C03679=1100.327,-122.776,-46.976,-179.986,4.175,148.668
C03680=1100.332,-123.026,-46.967,-179.985,4.170,148.666
C03681=1100.338,-123.276,-46.957,-179.985,4.164,148.665
C03682=1100.343,-123.525,-46.946,-179.984,4.159,148.663
C03683=1100.348,-123.775,-46.938,-179.983,4.153,148.662
C03684=1100.353,-124.026,-46.927,-179.983,4.148,148.661
C03685=1100.358,-124.275,-46.917,-179.982,4.143,148.659
C03686=1100.364,-124.524,-46.907,-179.982,4.138,148.658
C03687=1100.369,-124.774,-46.898,-179.981,4.133,148.657
C03688=1100.375,-125.024,-46.888,-179.980,4.128,148.655
C03689=1100.380,-125.274,-46.877,-179.980,4.122,148.654
C03690=1100.385,-125.524,-46.869,-179.979,4.117,148.653
C03691=1100.390,-125.773,-46.858,-179.978,4.111,148.651
C03692=1100.395,-126.023,-46.849,-179.978,4.106,148.650
C03693=1100.401,-126.273,-46.839,-179.977,4.102,148.649
C03694=1100.406,-126.522,-46.830,-179.976,4.096,148.647
C03695=1100.410,-126.736,-46.821,-179.976,4.091,148.646
C03696=1100.415,-126.951,-46.813,-179.975,4.087,148.645
C03697=1100.419,-127.165,-46.805,-179.974,4.083,148.644
C03698=1100.424,-127.380,-46.796,-179.974,4.077,148.642
C03699=1100.428,-127.594,-46.788,-179.973,4.073,148.641
C03700=1100.433,-127.809,-46.780,-179.972,4.069,148.640
C03701=1100.437,-128.023,-46.771,-179.972,4.064,148.639
C03702=1100.442,-128.238,-46.763,-179.971,4.059,148.637
C03703=1100.019,-128.228,-46.789,-179.964,4.064,148.636
C03704=1100.015,-128.014,-46.798,-179.965,4.068,148.637
C03705=1100.010,-127.799,-46.806,-179.966,4.073,148.639
C03706=1100.006,-127.585,-46.814,-179.966,4.078,148.640
C03707=1100.001,-127.371,-46.823,-179.966,4.082,148.641
C03708=1099.997,-127.156,-46.831,-179.967,4.086,148.642
C03709=1099.992,-126.942,-46.839,-179.968,4.091,148.643
C03710=1099.987,-126.728,-46.847,-179.968,4.096,148.645
C03711=1099.983,-126.513,-46.856,-179.969,4.100,148.646
C03712=1099.978,-126.263,-46.866,-179.970,4.105,148.647
C03713=1099.972,-126.013,-46.875,-179.970,4.111,148.649
C03714=1099.967,-125.764,-46.885,-179.971,4.116,148.650
C03715=1099.962,-125.515,-46.895,-179.972,4.121,148.651
C03716=1099.956,-125.264,-46.904,-179.972,4.127,148.653
C03717=1099.952,-125.014,-46.914,-179.973,4.131,148.654
C03718=1099.946,-124.765,-46.925,-179.974,4.137,148.655
C03719=1099.941,-124.515,-46.933,-179.974,4.142,148.657
C03720=1099.935,-124.266,-46.944,-179.975,4.147,148.658
C03721=1099.930,-124.016,-46.954,-179.976,4.153,148.660
C03722=1099.926,-123.766,-46.964,-179.976,4.158,148.661
C03723=1099.920,-123.516,-46.973,-179.977,4.164,148.662
C03724=1099.915,-123.267,-46.983,-179.978,4.168,148.663
C03725=1099.909,-123.017,-46.993,-179.979,4.173,148.665
C03726=1099.904,-122.766,-47.003,-179.979,4.179,148.666
C03727=1099.899,-122.517,-47.013,-179.980,4.184,148.668
C03728=1099.894,-122.267,-47.023,-179.980,4.189,148.669
C03729=1099.888,-122.018,-47.033,-179.982,4.194,148.670
C03730=1099.884,-121.768,-47.043,-179.982,4.199,148.672
C03731=1099.878,-121.518,-47.053,-179.983,4.205,148.673
C03732=1099.873,-121.269,-47.062,-179.983,4.210,148.674
C03733=1099.867,-121.019,-47.072,-179.984,4.215,148.676
C03734=1099.862,-120.769,-47.083,-179.984,4.220,148.677
C03735=1099.857,-120.520,-47.093,-179.985,4.225,148.678
C03736=1099.852,-120.269,-47.102,-179.986,4.230,148.680
C03737=1099.846,-120.020,-47.112,-179.986,4.235,148.681
C03738=1099.842,-119.770,-47.122,-179.987,4.241,148.682
C03739=1099.836,-119.520,-47.132,-179.987,4.246,148.683
C03740=1099.830,-119.271,-47.143,-179.988,4.251,148.685
C03741=1099.826,-119.021,-47.153,-179.989,4.256,148.686
C03742=1099.820,-118.771,-47.162,-179.989,4.261,148.687
C03743=1099.815,-118.521,-47.172,-179.990,4.267,148.689
C03744=1099.810,-118.271,-47.183,-179.991,4.271,148.690
C03745=1099.805,-118.022,-47.193,-179.991,4.277,148.692
C03746=1099.799,-117.772,-47.203,-179.992,4.282,148.693
C03747=1099.794,-117.523,-47.213,-179.992,4.287,148.694
C03748=1099.789,-117.272,-47.224,-179.993,4.292,148.695
C03749=1099.784,-117.023,-47.233,-179.994,4.297,148.697
C03750=1099.778,-116.774,-47.243,-179.994,4.302,148.698
C03751=1099.773,-116.523,-47.253,-179.995,4.307,148.699
C03752=1099.767,-116.273,-47.263,-179.995,4.313,148.701
C03753=1099.762,-116.024,-47.273,-179.996,4.317,148.702
C03754=1099.757,-115.774,-47.284,-179.997,4.322,148.703
C03755=1099.752,-115.524,-47.294,-179.997,4.328,148.704
C03756=1099.746,-115.275,-47.304,-179.997,4.333,148.706
C03757=1099.742,-115.025,-47.314,-179.998,4.337,148.707
C03758=1099.736,-114.775,-47.324,-179.999,4.343,148.708
C03759=1099.731,-114.526,-47.334,-179.999,4.348,148.710
C03760=1099.727,-114.312,-47.343,-180.000,4.352,148.711
C03761=1099.722,-114.097,-47.352,180.000,4.356,148.712
C03762=1099.717,-113.882,-47.361,180.000,4.361,148.713
C03763=1099.713,-113.668,-47.370,179.999,4.365,148.714
C03764=1099.709,-113.454,-47.378,179.998,4.369,148.715
C03765=1099.705,-113.240,-47.387,179.998,4.374,148.716
C03766=1099.700,-113.025,-47.396,179.997,4.378,148.717
C03767=1099.695,-112.811,-47.405,179.997,4.383,148.718
C03768=1099.690,-112.562,-47.415,179.996,4.387,148.720
C03769=1099.685,-112.312,-47.426,179.996,4.392,148.721
C03770=1099.680,-112.062,-47.436,179.996,4.398,148.722
C03771=1099.674,-111.813,-47.446,179.995,4.403,148.724
C03772=1099.669,-111.562,-47.457,179.994,4.407,148.725
C03773=1099.663,-111.313,-47.467,179.994,4.413,148.726
C03774=1099.658,-111.062,-47.477,179.994,4.418,148.727
C03775=1099.654,-110.813,-47.487,179.992,4.422,148.729
C03776=1099.648,-110.564,-47.497,179.992,4.428,148.730
C03777=1099.643,-110.313,-47.508,179.992,4.433,148.731
C03778=1099.637,-110.064,-47.518,179.991,4.438,148.732
C03779=1099.633,-109.814,-47.529,179.991,4.442,148.734
C03780=1099.627,-109.565,-47.540,179.990,4.448,148.735
C03781=1099.621,-109.315,-47.550,179.990,4.453,148.736
C03782=1099.616,-109.065,-47.560,179.989,4.457,148.737
C03783=1099.611,-108.815,-47.571,179.989,4.462,148.739
C03784=1099.607,-108.565,-47.581,179.988,4.467,148.740
C03785=1099.601,-108.316,-47.591,179.988,4.473,148.741
C03786=1099.596,-108.066,-47.602,179.987,4.477,148.742
C03787=1099.591,-107.817,-47.612,179.986,4.482,148.744
C03788=1099.586,-107.567,-47.623,179.986,4.488,148.745
C03789=1099.580,-107.317,-47.633,179.985,4.492,148.746
C03790=1099.575,-107.067,-47.643,179.985,4.497,148.747
C03791=1099.570,-106.817,-47.654,179.984,4.503,148.749
C03792=1099.564,-106.568,-47.665,179.984,4.508,148.750
C03793=1099.559,-106.318,-47.675,179.983,4.512,148.751
C03794=1099.554,-106.068,-47.685,179.983,4.517,148.752
C03795=1099.549,-105.818,-47.696,179.983,4.522,148.754
C03796=1099.543,-105.569,-47.707,179.982,4.527,148.755
C03797=1099.538,-105.319,-47.718,179.982,4.532,148.756
C03798=1099.533,-105.070,-47.728,179.981,4.537,148.757
C03799=1099.528,-104.819,-47.738,179.980,4.542,148.759
C03800=1099.522,-104.570,-47.749,179.980,4.547,148.760
C03801=1099.517,-104.320,-47.760,179.980,4.552,148.761
C03802=1099.512,-104.071,-47.770,179.979,4.556,148.762
C03803=1099.507,-103.820,-47.781,179.979,4.561,148.763
C03804=1099.502,-103.571,-47.792,179.979,4.567,148.765
C03805=1099.497,-103.321,-47.802,179.978,4.571,148.766
C03806=1099.491,-103.072,-47.812,179.977,4.576,148.767
C03807=1099.486,-102.822,-47.824,179.977,4.582,148.768
C03808=1099.481,-102.572,-47.834,179.976,4.587,148.770
C03809=1099.476,-102.322,-47.844,179.976,4.591,148.771
C03810=1099.470,-102.073,-47.855,179.975,4.596,148.772
C03811=1099.465,-101.823,-47.866,179.975,4.601,148.773
C03812=1099.460,-101.573,-47.876,179.974,4.606,148.774
C03813=1099.455,-101.324,-47.887,179.974,4.611,148.776
C03814=1099.450,-101.074,-47.898,179.974,4.616,148.777
C03815=1099.445,-100.825,-47.909,179.973,4.620,148.778
C03816=1099.440,-100.610,-47.918,179.972,4.625,148.779
C03817=1099.435,-100.396,-47.927,179.973,4.629,148.780
C03818=1099.432,-100.182,-47.936,179.972,4.633,148.781
C03819=1099.427,-99.967,-47.946,179.972,4.638,148.782
C03820=1099.423,-99.754,-47.955,179.971,4.642,148.783
C03821=1099.417,-99.539,-47.964,179.971,4.646,148.784
C03822=1099.413,-99.325,-47.973,179.970,4.650,148.786
C03823=1099.409,-99.110,-47.983,179.970,4.654,148.786
C03824=1099.403,-98.861,-47.993,179.970,4.659,148.788
C03825=1099.399,-98.611,-48.004,179.969,4.664,148.789
C03826=1099.393,-98.361,-48.015,179.969,4.668,148.790
C03827=1099.388,-98.112,-48.026,179.968,4.674,148.791
C03828=1099.383,-97.862,-48.036,179.968,4.679,148.792
C03829=1099.378,-97.613,-48.047,179.967,4.683,148.794
C03830=1099.372,-97.362,-48.059,179.967,4.688,148.795
C03831=1099.367,-97.113,-48.070,179.967,4.693,148.796
C03832=1099.362,-96.863,-48.080,179.966,4.698,148.797
C03833=1099.357,-96.614,-48.091,179.965,4.703,148.799
C03834=1099.352,-96.364,-48.102,179.965,4.708,148.800
C03835=1099.347,-96.114,-48.113,179.964,4.713,148.801
C03836=1099.341,-95.864,-48.123,179.964,4.718,148.802
C03837=1099.336,-95.615,-48.135,179.964,4.723,148.804
C03838=1099.330,-95.365,-48.145,179.963,4.727,148.805
C03839=1099.326,-95.115,-48.156,179.963,4.732,148.806
C03840=1099.321,-94.865,-48.167,179.963,4.738,148.807
C03841=1099.315,-94.616,-48.178,179.962,4.742,148.808
C03842=1099.310,-94.366,-48.189,179.962,4.747,148.809
C03843=1099.305,-94.116,-48.200,179.962,4.752,148.811
C03844=1099.300,-93.867,-48.211,179.961,4.757,148.812
C03845=1099.295,-93.617,-48.222,179.961,4.762,148.813
C03846=1099.289,-93.367,-48.234,179.960,4.767,148.814
C03847=1099.284,-93.117,-48.244,179.960,4.772,148.815
C03848=1099.279,-92.868,-48.255,179.960,4.777,148.817
C03849=1099.273,-92.618,-48.266,179.959,4.781,148.818
C03850=1099.269,-92.369,-48.277,179.959,4.787,148.819
C03851=1099.263,-92.119,-48.289,179.959,4.792,148.820
C03852=1099.258,-91.868,-48.299,179.959,4.797,148.821
C03853=1099.253,-91.619,-48.310,179.959,4.802,148.823
C03854=1099.248,-91.370,-48.322,179.958,4.806,148.824
C03855=1099.243,-91.119,-48.333,179.958,4.811,148.825
C03856=1099.237,-90.870,-48.344,179.957,4.817,148.826
C03857=1099.233,-90.621,-48.355,179.957,4.822,148.827
C03858=1099.227,-90.370,-48.366,179.957,4.827,148.829
C03859=1099.222,-90.121,-48.377,179.957,4.832,148.830
C03860=1099.217,-89.872,-48.388,179.956,4.836,148.831
C03861=1099.211,-89.621,-48.399,179.956,4.841,148.832
C03862=1099.206,-89.372,-48.410,179.956,4.847,148.833
C03863=1099.201,-89.123,-48.422,179.955,4.852,148.835
C03864=1099.196,-88.873,-48.433,179.955,4.857,148.836
C03865=1099.191,-88.622,-48.444,179.955,4.862,148.837
C03866=1099.185,-88.373,-48.455,179.955,4.867,148.838
C03867=1099.181,-88.124,-48.466,179.954,4.871,148.839
C03868=1099.175,-87.874,-48.478,179.954,4.877,148.840
C03869=1099.170,-87.624,-48.489,179.954,4.882,148.842
C03870=1099.164,-87.374,-48.500,179.954,4.887,148.843
C03871=1099.160,-87.125,-48.512,179.953,4.892,148.844
C03872=1099.155,-86.869,-48.523,179.953,4.897,148.845
C03873=1099.149,-86.613,-48.534,179.952,4.903,148.847
C03874=1099.144,-86.358,-48.546,179.952,4.908,148.848
C03875=1099.138,-86.102,-48.558,179.952,4.913,148.849
C03876=1099.134,-85.853,-48.569,179.952,4.918,148.850
C03877=1099.128,-85.603,-48.581,179.952,4.923,148.851
C03878=1099.123,-85.354,-48.592,179.952,4.928,148.853
C03879=1099.118,-85.104,-48.603,179.951,4.933,148.854
C03880=1099.113,-84.854,-48.614,179.951,4.938,148.855
C03881=1099.108,-84.604,-48.626,179.950,4.943,148.856
C03882=1099.102,-84.355,-48.637,179.950,4.948,148.858
C03883=1099.097,-84.105,-48.648,179.950,4.954,148.859
C03884=1099.092,-83.856,-48.660,179.949,4.959,148.860
C03885=1099.087,-83.606,-48.672,179.949,4.964,148.861
C03886=1099.082,-83.356,-48.683,179.949,4.969,148.862
C03887=1099.076,-83.106,-48.694,179.949,4.974,148.863
C03888=1099.071,-82.856,-48.705,179.949,4.979,148.865
C03889=1099.066,-82.607,-48.717,179.948,4.984,148.866
C03890=1099.061,-82.357,-48.728,179.948,4.989,148.867
C03891=1099.056,-82.107,-48.740,179.947,4.994,148.868
C03892=1098.828,-91.515,-48.346,179.965,4.807,148.822
C03893=1098.834,-91.764,-48.335,179.965,4.802,148.821
C03894=1098.838,-92.013,-48.323,179.965,4.797,148.819
C03895=1098.844,-92.264,-48.312,179.966,4.793,148.818
C03896=1098.849,-92.513,-48.301,179.966,4.788,148.817
C03897=1098.854,-92.762,-48.290,179.966,4.782,148.816
C03898=1098.859,-93.013,-48.279,179.966,4.777,148.815
C03899=1098.865,-93.262,-48.268,179.967,4.772,148.814
C03900=1098.870,-93.512,-48.257,179.967,4.768,148.812
C03901=1098.875,-93.762,-48.246,179.968,4.763,148.811
C03902=1098.880,-94.011,-48.235,179.968,4.758,148.810
C03903=1098.886,-94.261,-48.224,179.968,4.752,148.809
C03904=1098.890,-94.511,-48.213,179.969,4.748,148.808
C03905=1098.896,-94.761,-48.202,179.969,4.743,148.806
C03906=1098.901,-95.010,-48.191,179.969,4.738,148.805
C03907=1098.907,-95.259,-48.180,179.970,4.733,148.804
C03908=1098.912,-95.510,-48.169,179.970,4.728,148.803
C03909=1098.916,-95.759,-48.158,179.970,4.723,148.802
C03910=1098.922,-96.009,-48.148,179.971,4.719,148.800
C03911=1098.927,-96.258,-48.136,179.971,4.714,148.799
C03912=1098.932,-96.509,-48.126,179.972,4.709,148.798
C03913=1098.938,-96.758,-48.114,179.972,4.704,148.797
C03914=1098.943,-97.008,-48.104,179.973,4.699,148.796
C03915=1098.948,-97.257,-48.093,179.973,4.694,148.794
C03916=1098.953,-97.507,-48.082,179.974,4.689,148.793
C03917=1098.958,-97.757,-48.071,179.974,4.684,148.792
C03918=1098.964,-98.007,-48.060,179.975,4.679,148.791
C03919=1098.969,-98.256,-48.049,179.975,4.675,148.789
C03920=1098.974,-98.506,-48.038,179.976,4.670,148.788
C03921=1098.979,-98.756,-48.027,179.976,4.664,148.787
C03922=1098.984,-99.006,-48.017,179.977,4.660,148.786
C03923=1098.989,-99.255,-48.006,179.977,4.655,148.785
C03924=1098.994,-99.505,-47.995,179.977,4.650,148.783
C03925=1099.001,-99.832,-47.981,179.978,4.644,148.782
C03926=1099.008,-100.160,-47.967,179.978,4.638,148.780
C03927=1099.015,-100.488,-47.953,179.979,4.631,148.779
C03928=1099.022,-100.815,-47.938,179.980,4.624,148.777
C03929=1099.028,-101.065,-47.928,179.981,4.620,148.776
C03930=1099.032,-101.315,-47.917,179.981,4.615,148.774
C03931=1099.038,-101.564,-47.906,179.981,4.609,148.773
C03932=1099.043,-101.814,-47.896,179.982,4.605,148.772
C03933=1099.048,-102.063,-47.885,179.982,4.600,148.771
C03934=1099.053,-102.313,-47.874,179.982,4.595,148.770
C03935=1099.058,-102.563,-47.863,179.983,4.591,148.768
C03936=1099.063,-102.813,-47.853,179.983,4.585,148.767
C03937=1099.069,-103.063,-47.842,179.984,4.580,148.766
C03938=1099.074,-103.312,-47.831,179.984,4.575,148.765
C03939=1099.079,-103.562,-47.820,179.985,4.570,148.763
C03940=1099.085,-103.812,-47.810,179.985,4.565,148.762
C03941=1099.090,-104.062,-47.799,179.986,4.560,148.761
C03942=1099.095,-104.311,-47.789,179.986,4.556,148.760
C03943=1099.100,-104.561,-47.778,179.987,4.551,148.759
C03944=1099.106,-104.811,-47.768,179.987,4.545,148.757
C03945=1099.111,-105.061,-47.756,179.988,4.541,148.756
C03946=1099.116,-105.310,-47.746,179.988,4.536,148.755
C03947=1099.121,-105.560,-47.736,179.989,4.530,148.754
C03948=1099.126,-105.809,-47.725,179.989,4.526,148.752
C03949=1099.131,-106.059,-47.714,179.990,4.521,148.751
C03950=1099.137,-106.309,-47.704,179.990,4.516,148.750
C03951=1099.142,-106.559,-47.693,179.991,4.512,148.749
C03952=1099.147,-106.808,-47.682,179.991,4.506,148.748
C03953=1099.152,-107.058,-47.673,179.992,4.501,148.746
C03954=1099.157,-107.308,-47.662,179.993,4.497,148.745
C03955=1099.162,-107.558,-47.652,179.993,4.491,148.744
C03956=1099.168,-107.807,-47.642,179.993,4.486,148.742
C03957=1099.173,-108.057,-47.630,179.993,4.481,148.741
C03958=1099.178,-108.307,-47.620,179.994,4.477,148.740
C03959=1099.183,-108.557,-47.609,179.995,4.471,148.739
C03960=1099.189,-108.806,-47.599,179.995,4.466,148.737
C03961=1099.194,-109.056,-47.589,179.996,4.462,148.736
C03962=1099.199,-109.306,-47.578,179.996,4.457,148.735
C03963=1099.205,-109.555,-47.568,179.996,4.451,148.734
C03964=1099.210,-109.805,-47.557,179.997,4.446,148.732
C03965=1099.215,-110.055,-47.547,179.998,4.442,148.731
C03966=1099.220,-110.305,-47.536,179.998,4.436,148.730
C03967=1099.225,-110.554,-47.527,179.999,4.431,148.729
C03968=1099.231,-110.804,-47.516,180.000,4.427,148.727
C03969=1099.235,-111.054,-47.505,-180.000,4.421,148.726
C03970=1099.241,-111.303,-47.495,-180.000,4.416,148.725
C03971=1099.246,-111.553,-47.484,-179.999,4.411,148.724
C03972=1099.252,-111.803,-47.474,-179.998,4.407,148.722
C03973=1099.257,-112.053,-47.463,-179.998,4.401,148.721
C03974=1099.262,-112.303,-47.453,-179.997,4.396,148.720
C03975=1099.267,-112.552,-47.444,-179.997,4.392,148.718
C03976=1099.272,-112.802,-47.433,-179.996,4.386,148.717
C03977=1099.276,-113.016,-47.424,-179.996,4.382,148.716
C03978=1099.281,-113.231,-47.415,-179.995,4.377,148.715
C03979=1099.286,-113.445,-47.406,-179.995,4.373,148.714
C03980=1099.290,-113.659,-47.398,-179.994,4.369,148.713
C03981=1099.294,-113.873,-47.389,-179.994,4.365,148.712
C03982=1099.300,-114.088,-47.380,-179.993,4.361,148.710
C03983=1099.304,-114.302,-47.371,-179.993,4.356,148.710
C03984=1099.308,-114.516,-47.362,-179.992,4.352,148.708
C03985=1099.314,-114.766,-47.352,-179.992,4.346,148.707
C03986=1099.319,-115.016,-47.342,-179.991,4.342,148.706
C03987=1099.324,-115.265,-47.332,-179.990,4.337,148.704
C03988=1099.329,-115.515,-47.321,-179.990,4.331,148.703
C03989=1099.334,-115.765,-47.311,-179.990,4.326,148.702
C03990=1099.340,-116.014,-47.301,-179.989,4.322,148.701
C03991=1099.345,-116.265,-47.290,-179.988,4.316,148.699
C03992=1099.350,-116.514,-47.281,-179.988,4.311,148.698
C03993=1099.355,-116.763,-47.271,-179.987,4.306,148.697
C03994=1099.360,-117.014,-47.260,-179.986,4.301,148.695
C03995=1099.366,-117.263,-47.250,-179.986,4.296,148.694
C03996=1099.371,-117.512,-47.240,-179.985,4.291,148.693
C03997=1099.376,-117.763,-47.230,-179.985,4.286,148.692
C03998=1099.382,-118.013,-47.220,-179.984,4.281,148.690
C03999=1099.387,-118.262,-47.210,-179.983,4.276,148.689
C04000=1099.392,-118.512,-47.200,-179.983,4.271,148.688
C04001=1099.397,-118.762,-47.190,-179.982,4.265,148.686
C04002=1099.403,-119.011,-47.180,-179.981,4.261,148.685
C04003=1099.408,-119.261,-47.169,-179.981,4.255,148.683
C04004=1099.413,-119.511,-47.159,-179.980,4.250,148.682
C04005=1099.418,-119.760,-47.149,-179.980,4.244,148.681
C04006=1099.424,-120.011,-47.140,-179.979,4.239,148.680
C04007=1099.428,-120.260,-47.130,-179.978,4.235,148.678
C04008=1099.434,-120.510,-47.119,-179.978,4.229,148.677
C04009=1099.440,-120.760,-47.109,-179.977,4.224,148.676
C04010=1099.444,-121.009,-47.099,-179.977,4.219,148.674
C04011=1099.449,-121.259,-47.089,-179.976,4.214,148.673
C04012=1099.455,-121.509,-47.080,-179.975,4.209,148.672
C04013=1099.460,-121.758,-47.070,-179.975,4.204,148.670
C04014=1099.465,-122.009,-47.059,-179.974,4.198,148.669
C04015=1099.471,-122.258,-47.049,-179.974,4.193,148.668
C04016=1099.476,-122.507,-47.040,-179.973,4.188,148.666
C04017=1099.482,-122.758,-47.030,-179.972,4.183,148.665
C04018=1099.487,-123.008,-47.020,-179.971,4.178,148.663
C04019=1099.491,-123.257,-47.010,-179.971,4.173,148.662
C04020=1099.497,-123.507,-47.000,-179.970,4.167,148.661
C04021=1099.502,-123.756,-46.991,-179.970,4.162,148.660
C04022=1099.507,-124.007,-46.980,-179.969,4.156,148.658
C04023=1099.513,-124.256,-46.970,-179.968,4.152,148.657
C04024=1099.518,-124.505,-46.960,-179.967,4.146,148.655
C04025=1099.524,-124.756,-46.951,-179.966,4.141,148.654
C04026=1099.528,-125.006,-46.941,-179.966,4.136,148.653
C04027=1099.533,-125.255,-46.931,-179.965,4.130,148.651
C04028=1099.539,-125.505,-46.921,-179.965,4.125,148.650
C04029=1099.544,-125.755,-46.912,-179.964,4.120,148.649
C04030=1099.550,-126.004,-46.901,-179.963,4.115,148.647
C04031=1099.554,-126.254,-46.891,-179.962,4.110,148.646
C04032=1099.560,-126.504,-46.882,-179.962,4.104,148.644
C04033=1099.564,-126.719,-46.874,-179.961,4.100,148.643
C04034=1099.569,-126.932,-46.865,-179.961,4.095,148.642
C04035=1099.573,-127.147,-46.856,-179.960,4.091,148.641
C04036=1099.578,-127.361,-46.848,-179.959,4.086,148.640
C04037=1099.582,-127.576,-46.840,-179.959,4.081,148.638
C04038=1099.587,-127.790,-46.832,-179.958,4.077,148.637
C04039=1099.592,-128.004,-46.823,-179.957,4.073,148.636
C04040=1099.596,-128.219,-46.815,-179.957,4.067,148.635
C04041=1099.173,-128.209,-46.841,-179.950,4.072,148.634
C04042=1099.168,-127.995,-46.849,-179.951,4.076,148.635
C04043=1099.164,-127.781,-46.858,-179.951,4.082,148.636
C04044=1099.160,-127.567,-46.866,-179.952,4.086,148.637
C04045=1099.155,-127.352,-46.874,-179.952,4.090,148.638
C04046=1099.151,-127.138,-46.883,-179.952,4.095,148.639
C04047=1099.146,-126.923,-46.891,-179.953,4.099,148.641
C04048=1099.142,-126.709,-46.899,-179.954,4.104,148.642
C04049=1099.137,-126.494,-46.908,-179.954,4.109,148.643
C04050=1099.131,-126.245,-46.918,-179.955,4.113,148.644
C04051=1099.127,-125.996,-46.927,-179.956,4.119,148.646
C04052=1099.122,-125.745,-46.938,-179.957,4.124,148.647
C04053=1099.116,-125.495,-46.947,-179.957,4.129,148.649
C04054=1099.111,-125.246,-46.957,-179.958,4.135,148.650
C04055=1099.105,-124.996,-46.967,-179.958,4.140,148.651
C04056=1099.101,-124.746,-46.976,-179.960,4.145,148.653
C04057=1099.095,-124.496,-46.987,-179.961,4.150,148.654
C04058=1099.089,-124.247,-46.997,-179.961,4.156,148.655
C04059=1099.085,-123.997,-47.007,-179.962,4.161,148.657
C04060=1099.080,-123.747,-47.017,-179.962,4.166,148.658
C04061=1099.074,-123.497,-47.027,-179.963,4.172,148.660
C04062=1099.069,-123.248,-47.036,-179.964,4.176,148.661
C04063=1099.063,-122.998,-47.046,-179.964,4.182,148.662
C04064=1099.058,-122.748,-47.057,-179.965,4.187,148.663
C04065=1099.053,-122.498,-47.066,-179.966,4.192,148.665
C04066=1099.047,-122.249,-47.076,-179.966,4.198,148.666
C04067=1099.042,-121.999,-47.086,-179.967,4.202,148.668
C04068=1099.038,-121.749,-47.096,-179.968,4.208,148.669
C04069=1099.032,-121.500,-47.106,-179.968,4.213,148.670
C04070=1099.026,-121.250,-47.117,-179.969,4.218,148.672
C04071=1099.022,-121.000,-47.126,-179.969,4.223,148.673
C04072=1099.016,-120.750,-47.136,-179.970,4.228,148.674
C04073=1099.011,-120.500,-47.146,-179.971,4.233,148.676
C04074=1099.006,-120.251,-47.156,-179.971,4.238,148.677
C04075=1099.001,-120.001,-47.167,-179.972,4.244,148.678
C04076=1098.995,-119.751,-47.177,-179.972,4.249,148.680
C04077=1098.990,-119.502,-47.186,-179.974,4.254,148.681
C04078=1098.985,-119.252,-47.197,-179.974,4.259,148.682
C04079=1098.980,-119.002,-47.207,-179.975,4.265,148.684
C04080=1098.974,-118.752,-47.217,-179.975,4.270,148.685
C04081=1098.970,-118.502,-47.227,-179.976,4.274,148.686
C04082=1098.964,-118.253,-47.237,-179.977,4.280,148.688
C04083=1098.958,-118.003,-47.247,-179.977,4.285,148.689
C04084=1098.953,-117.753,-47.258,-179.978,4.290,148.690
C04085=1098.949,-117.504,-47.267,-179.978,4.295,148.692
C04086=1098.943,-117.254,-47.277,-179.979,4.300,148.693
C04087=1098.938,-117.004,-47.288,-179.980,4.305,148.694
C04088=1098.932,-116.754,-47.298,-179.980,4.310,148.695
C04089=1098.927,-116.505,-47.308,-179.980,4.316,148.697
C04090=1098.922,-116.255,-47.318,-179.982,4.320,148.698
C04091=1098.917,-116.005,-47.329,-179.982,4.325,148.699
C04092=1098.911,-115.756,-47.339,-179.982,4.331,148.701
C04093=1098.906,-115.506,-47.349,-179.983,4.336,148.702
C04094=1098.901,-115.256,-47.360,-179.984,4.340,148.703
C04095=1098.896,-115.006,-47.370,-179.984,4.346,148.704
C04096=1098.891,-114.757,-47.380,-179.985,4.351,148.706
C04097=1098.885,-114.507,-47.390,-179.986,4.355,148.707
C04098=1098.877,-114.095,-47.407,-179.986,4.364,148.709
C04099=1098.868,-113.684,-47.424,-179.987,4.373,148.711
C04100=1098.860,-113.273,-47.441,-179.988,4.381,148.713
C04101=1098.850,-112.861,-47.458,-179.989,4.389,148.716
C04102=1098.846,-112.611,-47.468,-179.990,4.394,148.717
C04103=1098.841,-112.362,-47.479,-179.990,4.398,148.718
C04104=1098.835,-112.112,-47.489,-179.991,4.404,148.719
C04105=1098.830,-111.862,-47.500,-179.991,4.409,148.721
C04106=1098.825,-111.613,-47.510,-179.992,4.414,148.722
C04107=1098.819,-111.363,-47.520,-179.993,4.419,148.723
C04108=1098.814,-111.113,-47.531,-179.993,4.424,148.725
C04109=1098.809,-110.863,-47.541,-179.994,4.429,148.726
C04110=1098.804,-110.613,-47.552,-179.994,4.434,148.727
C04111=1098.799,-110.364,-47.562,-179.995,4.439,148.728
C04112=1098.794,-110.114,-47.573,-179.995,4.444,148.730
C04113=1098.788,-109.865,-47.583,-179.996,4.449,148.731
C04114=1098.783,-109.614,-47.593,-179.996,4.454,148.732
C04115=1098.778,-109.365,-47.604,-179.997,4.459,148.733
C04116=1098.772,-109.115,-47.614,-179.997,4.464,148.734
C04117=1098.768,-108.866,-47.625,-179.998,4.469,148.736
C04118=1098.762,-108.616,-47.635,-179.999,4.474,148.737
C04119=1098.757,-108.366,-47.646,-179.999,4.479,148.738
C04120=1098.751,-108.116,-47.656,-179.999,4.484,148.740
C04121=1098.747,-107.867,-47.667,-180.000,4.489,148.741
C04122=1098.741,-107.617,-47.678,179.999,4.494,148.742
C04123=1098.736,-107.367,-47.688,179.999,4.499,148.743
C04124=1098.730,-107.117,-47.698,179.998,4.504,148.745
C04125=1098.725,-106.867,-47.709,179.998,4.509,148.746
C04126=1098.720,-106.618,-47.720,179.998,4.514,148.747
C04127=1098.715,-106.368,-47.730,179.997,4.518,148.748
C04128=1098.710,-106.118,-47.741,179.996,4.524,148.750
C04129=1098.705,-105.869,-47.752,179.996,4.529,148.751
C04130=1098.699,-105.619,-47.762,179.995,4.533,148.752
C04131=1098.694,-105.369,-47.773,179.995,4.538,148.753
C04132=1098.689,-105.119,-47.783,179.995,4.543,148.755
C04133=1098.684,-104.870,-47.794,179.994,4.548,148.756
C04134=1098.678,-104.620,-47.804,179.994,4.553,148.757
C04135=1098.673,-104.370,-47.815,179.993,4.558,148.758
C04136=1098.668,-104.121,-47.826,179.992,4.563,148.760
C04137=1098.663,-103.871,-47.836,179.992,4.568,148.761
C04138=1098.657,-103.621,-47.847,179.992,4.573,148.762
C04139=1098.653,-103.372,-47.858,179.991,4.578,148.763
C04140=1098.648,-103.121,-47.869,179.991,4.583,148.764
C04141=1098.643,-102.872,-47.879,179.990,4.588,148.766
C04142=1098.638,-102.622,-47.890,179.990,4.593,148.767
C04143=1098.632,-102.373,-47.900,179.989,4.597,148.768
C04144=1098.627,-102.123,-47.911,179.989,4.603,148.769
C04145=1098.622,-101.873,-47.922,179.988,4.608,148.771
C04146=1098.617,-101.623,-47.932,179.988,4.612,148.772
C04147=1098.611,-101.374,-47.943,179.987,4.617,148.773
C04148=1098.606,-101.124,-47.954,179.987,4.622,148.774
C04149=1098.601,-100.874,-47.966,179.986,4.627,148.775
C04150=1098.373,-110.205,-47.597,-179.988,4.446,148.728
C04151=1098.378,-110.455,-47.586,-179.988,4.441,148.726
C04152=1098.383,-110.704,-47.575,-179.987,4.436,148.725
C04153=1098.389,-110.954,-47.565,-179.987,4.431,148.724
C04154=1098.394,-111.204,-47.555,-179.986,4.426,148.723
C04155=1098.399,-111.453,-47.545,-179.985,4.421,148.721
C04156=1098.404,-111.703,-47.534,-179.985,4.416,148.720
C04157=1098.409,-111.953,-47.524,-179.984,4.411,148.719
C04158=1098.414,-112.203,-47.513,-179.984,4.406,148.718
C04159=1098.420,-112.452,-47.503,-179.983,4.401,148.716
C04160=1098.425,-112.702,-47.492,-179.983,4.396,148.715
C04161=1098.430,-112.952,-47.482,-179.982,4.391,148.714
C04162=1098.436,-113.201,-47.472,-179.981,4.386,148.712
C04163=1098.442,-113.526,-47.458,-179.981,4.379,148.711
C04164=1098.449,-113.849,-47.445,-179.981,4.373,148.709
C04165=1098.456,-114.174,-47.431,-179.979,4.367,148.708
C04166=1098.463,-114.497,-47.418,-179.979,4.360,148.706
C04167=1098.468,-114.748,-47.407,-179.978,4.355,148.705
C04168=1098.473,-114.997,-47.397,-179.978,4.349,148.703
C04169=1098.478,-115.246,-47.388,-179.977,4.345,148.702
C04170=1098.483,-115.497,-47.377,-179.976,4.340,148.701
C04171=1098.489,-115.746,-47.367,-179.976,4.334,148.699
C04172=1098.494,-115.996,-47.357,-179.975,4.329,148.698
C04173=1098.499,-116.246,-47.346,-179.975,4.325,148.697
C04174=1098.504,-116.495,-47.336,-179.974,4.319,148.695
C04175=1098.509,-116.746,-47.326,-179.973,4.314,148.694
C04176=1098.515,-116.995,-47.316,-179.973,4.309,148.693
C04177=1098.520,-117.245,-47.305,-179.972,4.304,148.692
C04178=1098.525,-117.495,-47.295,-179.972,4.299,148.690
C04179=1098.530,-117.744,-47.285,-179.971,4.294,148.689
C04180=1098.536,-117.994,-47.275,-179.970,4.289,148.688
C04181=1098.541,-118.244,-47.264,-179.970,4.284,148.686
C04182=1098.546,-118.493,-47.254,-179.969,4.279,148.685
C04183=1098.552,-118.743,-47.244,-179.969,4.274,148.684
C04184=1098.556,-118.993,-47.234,-179.968,4.268,148.682
C04185=1098.562,-119.242,-47.224,-179.967,4.264,148.681
C04186=1098.568,-119.492,-47.214,-179.966,4.258,148.680
C04187=1098.573,-119.742,-47.203,-179.966,4.253,148.678
C04188=1098.577,-119.991,-47.193,-179.966,4.248,148.677
C04189=1098.583,-120.241,-47.183,-179.965,4.242,148.676
C04190=1098.588,-120.492,-47.173,-179.964,4.238,148.674
C04191=1098.593,-120.741,-47.164,-179.963,4.232,148.673
C04192=1098.599,-120.991,-47.154,-179.963,4.227,148.672
C04193=1098.604,-121.241,-47.143,-179.962,4.222,148.670
C04194=1098.609,-121.490,-47.133,-179.961,4.217,148.669
C04195=1098.614,-121.740,-47.123,-179.960,4.212,148.668
C04196=1098.620,-121.989,-47.113,-179.960,4.207,148.666
C04197=1098.625,-122.239,-47.102,-179.959,4.201,148.665
C04198=1098.630,-122.489,-47.094,-179.959,4.196,148.664
C04199=1098.636,-122.739,-47.083,-179.958,4.191,148.662
C04200=1098.641,-122.989,-47.073,-179.957,4.186,148.661
C04201=1098.645,-123.238,-47.063,-179.956,4.181,148.660
C04202=1098.651,-123.488,-47.053,-179.956,4.176,148.658
C04203=1098.657,-123.738,-47.043,-179.955,4.170,148.657
C04204=1098.661,-123.988,-47.033,-179.954,4.165,148.655
C04205=1098.667,-124.237,-47.023,-179.954,4.160,148.654
C04206=1098.672,-124.487,-47.013,-179.953,4.155,148.653
C04207=1098.677,-124.737,-47.003,-179.953,4.150,148.651
C04208=1098.683,-124.987,-46.994,-179.952,4.144,148.650
C04209=1098.688,-125.237,-46.983,-179.951,4.138,148.649
C04210=1098.693,-125.486,-46.974,-179.950,4.134,148.647
C04211=1098.698,-125.736,-46.963,-179.949,4.129,148.646
C04212=1098.703,-125.986,-46.954,-179.949,4.123,148.645
C04213=1098.709,-126.236,-46.944,-179.948,4.118,148.643
C04214=1098.714,-126.485,-46.934,-179.947,4.112,148.642
C04215=1098.719,-126.700,-46.926,-179.947,4.108,148.641
C04216=1098.723,-126.914,-46.917,-179.946,4.104,148.639
C04217=1098.728,-127.128,-46.909,-179.946,4.099,148.638
C04218=1098.732,-127.342,-46.900,-179.945,4.095,148.637
C04219=1098.737,-127.557,-46.891,-179.944,4.090,148.636
C04220=1098.741,-127.771,-46.883,-179.944,4.085,148.635
C04221=1098.746,-127.986,-46.875,-179.943,4.081,148.633
C04222=1098.750,-128.200,-46.866,-179.942,4.076,148.632
C04223=1098.327,-128.190,-46.892,-179.935,4.080,148.631
C04224=1098.322,-127.977,-46.901,-179.936,4.085,148.632
C04225=1098.318,-127.763,-46.910,-179.937,4.090,148.633
C04226=1098.313,-127.550,-46.918,-179.937,4.094,148.635
C04227=1098.309,-127.337,-46.926,-179.937,4.099,148.636
C04228=1098.305,-127.123,-46.935,-179.938,4.103,148.637
C04229=1098.300,-126.909,-46.943,-179.939,4.108,148.638
C04230=1098.296,-126.696,-46.951,-179.940,4.112,148.639
C04231=1098.291,-126.483,-46.960,-179.940,4.117,148.640
C04232=1098.286,-126.233,-46.970,-179.940,4.122,148.642
C04233=1098.281,-125.984,-46.980,-179.942,4.127,148.643
C04234=1098.275,-125.734,-46.989,-179.943,4.132,148.645
C04235=1098.270,-125.483,-47.000,-179.943,4.138,148.646
C04236=1098.265,-125.234,-47.009,-179.944,4.143,148.647
C04237=1098.260,-124.985,-47.020,-179.945,4.149,148.649
C04238=1098.254,-124.734,-47.029,-179.945,4.154,148.650
C04239=1098.249,-124.484,-47.039,-179.946,4.159,148.651
C04240=1098.244,-124.235,-47.049,-179.947,4.164,148.653
C04241=1098.238,-123.985,-47.060,-179.947,4.169,148.654
C04242=1098.234,-123.735,-47.070,-179.948,4.174,148.655
C04243=1098.228,-123.486,-47.080,-179.948,4.180,148.657
C04244=1098.222,-123.236,-47.089,-179.950,4.185,148.658
C04245=1098.218,-122.987,-47.099,-179.950,4.190,148.660
C04246=1098.213,-122.736,-47.109,-179.951,4.195,148.661
C04247=1098.207,-122.487,-47.120,-179.951,4.200,148.662
C04248=1098.202,-122.238,-47.129,-179.952,4.206,148.664
C04249=1098.197,-121.987,-47.140,-179.953,4.210,148.665
C04250=1098.192,-121.738,-47.150,-179.954,4.216,148.666
C04251=1098.187,-121.488,-47.160,-179.954,4.221,148.668
C04252=1098.181,-121.238,-47.170,-179.955,4.226,148.669
C04253=1098.176,-120.988,-47.180,-179.956,4.231,148.670
C04254=1098.170,-120.739,-47.190,-179.956,4.236,148.672
C04255=1098.166,-120.489,-47.200,-179.957,4.241,148.673
C04256=1098.160,-120.239,-47.210,-179.958,4.247,148.674
C04257=1098.155,-119.990,-47.220,-179.958,4.252,148.676
C04258=1098.150,-119.739,-47.231,-179.959,4.257,148.677
C04259=1098.145,-119.490,-47.241,-179.960,4.262,148.678
C04260=1072.050,-72.101,295.701,-179.960,4.262,148.678
///USER 0
///POSTYPE ROBOT
///RECTAN
C04261=725.000,0.000,388.500,-180.000,-0.000,0.000
//INST
///DATE 2021/06/25 14:34
///ATTR SC,RW,RJ
////FRAME ROBOT
///GROUP1 RB1
NOP
MOVL C00000 V=800.0 PL=0
MOVL C00001 V=800.0 PL=0
MOVL C00002 V=800.0 PL=0
MOVL C00003 V=800.0 PL=0
MOVL C00004 V=800.0 PL=0
MOVL C00005 V=800.0 PL=0
MOVL C00006 V=800.0 PL=0
MOVL C00007 V=800.0 PL=0
MOVL C00008 V=800.0 PL=0
MOVL C00009 V=800.0 PL=0
MOVL C00010 V=800.0 PL=0
MOVL C00011 V=800.0 PL=0
MOVL C00012 V=800.0 PL=0
MOVL C00013 V=800.0 PL=0
MOVL C00014 V=800.0 PL=0
MOVL C00015 V=800.0 PL=0
MOVL C00016 V=800.0 PL=0
MOVL C00017 V=800.0 PL=0
MOVL C00018 V=800.0 PL=0
MOVL C00019 V=800.0 PL=0
MOVL C00020 V=800.0 PL=0
MOVL C00021 V=800.0 PL=0
MOVL C00022 V=800.0 PL=0
MOVL C00023 V=800.0 PL=0
MOVL C00024 V=800.0 PL=0
MOVL C00025 V=800.0 PL=0
MOVL C00026 V=800.0 PL=0
MOVL C00027 V=800.0 PL=0
MOVL C00028 V=800.0 PL=0
MOVL C00029 V=800.0 PL=0
MOVL C00030 V=800.0 PL=0
MOVL C00031 V=800.0 PL=0
MOVL C00032 V=800.0 PL=0
MOVL C00033 V=800.0 PL=0
MOVL C00034 V=800.0 PL=0
MOVL C00035 V=800.0 PL=0
MOVL C00036 V=800.0 PL=0
MOVL C00037 V=800.0 PL=0
MOVL C00038 V=800.0 PL=0
MOVL C00039 V=800.0 PL=0
MOVL C00040 V=800.0 PL=0
MOVL C00041 V=800.0 PL=0
MOVL C00042 V=800.0 PL=0
MOVL C00043 V=800.0 PL=0
MOVL C00044 V=800.0 PL=0
MOVL C00045 V=800.0 PL=0
MOVL C00046 V=800.0 PL=0
MOVL C00047 V=800.0 PL=0
MOVL C00048 V=800.0 PL=0
MOVL C00049 V=800.0 PL=0
MOVL C00050 V=800.0 PL=0
MOVL C00051 V=800.0 PL=0
MOVL C00052 V=800.0 PL=0
MOVL C00053 V=800.0 PL=0
MOVL C00054 V=800.0 PL=0
MOVL C00055 V=800.0 PL=0
MOVL C00056 V=800.0 PL=0
MOVL C00057 V=800.0 PL=0
MOVL C00058 V=800.0 PL=0
MOVL C00059 V=800.0 PL=0
MOVL C00060 V=800.0 PL=0
MOVL C00061 V=800.0 PL=0
MOVL C00062 V=800.0 PL=0
MOVL C00063 V=800.0 PL=0
MOVL C00064 V=800.0 PL=0
MOVL C00065 V=800.0 PL=0
MOVL C00066 V=800.0 PL=0
MOVL C00067 V=800.0 PL=0
MOVL C00068 V=800.0 PL=0
MOVL C00069 V=800.0 PL=0
MOVL C00070 V=800.0 PL=0
MOVL C00071 V=800.0 PL=0
MOVL C00072 V=800.0 PL=0
MOVL C00073 V=800.0 PL=0
MOVL C00074 V=800.0 PL=0
MOVL C00075 V=800.0 PL=0
MOVL C00076 V=800.0 PL=0
MOVL C00077 V=800.0 PL=0
MOVL C00078 V=800.0 PL=0
MOVL C00079 V=800.0 PL=0
MOVL C00080 V=800.0 PL=0
MOVL C00081 V=800.0 PL=0
MOVL C00082 V=800.0 PL=0
MOVL C00083 V=800.0 PL=0
MOVL C00084 V=800.0 PL=0
MOVL C00085 V=800.0 PL=0
MOVL C00086 V=800.0 PL=0
MOVL C00087 V=800.0 PL=0
MOVL C00088 V=800.0 PL=0
MOVL C00089 V=800.0 PL=0
MOVL C00090 V=800.0 PL=0
MOVL C00091 V=800.0 PL=0
MOVL C00092 V=800.0 PL=0
MOVL C00093 V=800.0 PL=0
MOVL C00094 V=800.0 PL=0
MOVL C00095 V=800.0 PL=0
MOVL C00096 V=800.0 PL=0
MOVL C00097 V=800.0 PL=0
MOVL C00098 V=800.0 PL=0
MOVL C00099 V=800.0 PL=0
MOVL C00100 V=800.0 PL=0
MOVL C00101 V=800.0 PL=0
MOVL C00102 V=800.0 PL=0
MOVL C00103 V=800.0 PL=0
MOVL C00104 V=800.0 PL=0
MOVL C00105 V=800.0 PL=0
MOVL C00106 V=800.0 PL=0
MOVL C00107 V=800.0 PL=0
MOVL C00108 V=800.0 PL=0
MOVL C00109 V=800.0 PL=0
MOVL C00110 V=800.0 PL=0
MOVL C00111 V=800.0 PL=0
MOVL C00112 V=800.0 PL=0
MOVL C00113 V=800.0 PL=0
MOVL C00114 V=800.0 PL=0
MOVL C00115 V=800.0 PL=0
MOVL C00116 V=800.0 PL=0
MOVL C00117 V=800.0 PL=0
MOVL C00118 V=800.0 PL=0
MOVL C00119 V=800.0 PL=0
MOVL C00120 V=800.0 PL=0
MOVL C00121 V=800.0 PL=0
MOVL C00122 V=800.0 PL=0
MOVL C00123 V=800.0 PL=0
MOVL C00124 V=800.0 PL=0
MOVL C00125 V=800.0 PL=0
MOVL C00126 V=800.0 PL=0
MOVL C00127 V=800.0 PL=0
MOVL C00128 V=800.0 PL=0
MOVL C00129 V=800.0 PL=0
MOVL C00130 V=800.0 PL=0
MOVL C00131 V=800.0 PL=0
MOVL C00132 V=800.0 PL=0
MOVL C00133 V=800.0 PL=0
MOVL C00134 V=800.0 PL=0
MOVL C00135 V=800.0 PL=0
MOVL C00136 V=800.0 PL=0
MOVL C00137 V=800.0 PL=0
MOVL C00138 V=800.0 PL=0
MOVL C00139 V=800.0 PL=0
MOVL C00140 V=800.0 PL=0
MOVL C00141 V=800.0 PL=0
MOVL C00142 V=800.0 PL=0
MOVL C00143 V=800.0 PL=0
MOVL C00144 V=800.0 PL=0
MOVL C00145 V=800.0 PL=0
MOVL C00146 V=800.0 PL=0
MOVL C00147 V=800.0 PL=0
MOVL C00148 V=800.0 PL=0
MOVL C00149 V=800.0 PL=0
MOVL C00150 V=800.0 PL=0
MOVL C00151 V=800.0 PL=0
MOVL C00152 V=800.0 PL=0
MOVL C00153 V=800.0 PL=0
MOVL C00154 V=800.0 PL=0
MOVL C00155 V=800.0 PL=0
MOVL C00156 V=800.0 PL=0
MOVL C00157 V=800.0 PL=0
MOVL C00158 V=800.0 PL=0
MOVL C00159 V=800.0 PL=0
MOVL C00160 V=800.0 PL=0
MOVL C00161 V=800.0 PL=0
MOVL C00162 V=800.0 PL=0
MOVL C00163 V=800.0 PL=0
MOVL C00164 V=800.0 PL=0
MOVL C00165 V=800.0 PL=0
MOVL C00166 V=800.0 PL=0
MOVL C00167 V=800.0 PL=0
MOVL C00168 V=800.0 PL=0
MOVL C00169 V=800.0 PL=0
MOVL C00170 V=800.0 PL=0
MOVL C00171 V=800.0 PL=0
MOVL C00172 V=800.0 PL=0
MOVL C00173 V=800.0 PL=0
MOVL C00174 V=800.0 PL=0
MOVL C00175 V=800.0 PL=0
MOVL C00176 V=800.0 PL=0
MOVL C00177 V=800.0 PL=0
MOVL C00178 V=800.0 PL=0
MOVL C00179 V=800.0 PL=0
MOVL C00180 V=800.0 PL=0
MOVL C00181 V=800.0 PL=0
MOVL C00182 V=800.0 PL=0
MOVL C00183 V=800.0 PL=0
MOVL C00184 V=800.0 PL=0
MOVL C00185 V=800.0 PL=0
MOVL C00186 V=800.0 PL=0
MOVL C00187 V=800.0 PL=0
MOVL C00188 V=800.0 PL=0
MOVL C00189 V=800.0 PL=0
MOVL C00190 V=800.0 PL=0
MOVL C00191 V=800.0 PL=0
MOVL C00192 V=800.0 PL=0
MOVL C00193 V=800.0 PL=0
MOVL C00194 V=800.0 PL=0
MOVL C00195 V=800.0 PL=0
MOVL C00196 V=800.0 PL=0
MOVL C00197 V=800.0 PL=0
MOVL C00198 V=800.0 PL=0
MOVL C00199 V=800.0 PL=0
MOVL C00200 V=800.0 PL=0
MOVL C00201 V=800.0 PL=0
MOVL C00202 V=800.0 PL=0
MOVL C00203 V=800.0 PL=0
MOVL C00204 V=800.0 PL=0
MOVL C00205 V=800.0 PL=0
MOVL C00206 V=800.0 PL=0
MOVL C00207 V=800.0 PL=0
MOVL C00208 V=800.0 PL=0
MOVL C00209 V=800.0 PL=0
MOVL C00210 V=800.0 PL=0
MOVL C00211 V=800.0 PL=0
MOVL C00212 V=800.0 PL=0
MOVL C00213 V=800.0 PL=0
MOVL C00214 V=800.0 PL=0
MOVL C00215 V=800.0 PL=0
MOVL C00216 V=800.0 PL=0
MOVL C00217 V=800.0 PL=0
MOVL C00218 V=800.0 PL=0
MOVL C00219 V=800.0 PL=0
MOVL C00220 V=800.0 PL=0
MOVL C00221 V=800.0 PL=0
MOVL C00222 V=800.0 PL=0
MOVL C00223 V=800.0 PL=0
MOVL C00224 V=800.0 PL=0
MOVL C00225 V=800.0 PL=0
MOVL C00226 V=800.0 PL=0
MOVL C00227 V=800.0 PL=0
MOVL C00228 V=800.0 PL=0
MOVL C00229 V=800.0 PL=0
MOVL C00230 V=800.0 PL=0
MOVL C00231 V=800.0 PL=0
MOVL C00232 V=800.0 PL=0
MOVL C00233 V=800.0 PL=0
MOVL C00234 V=800.0 PL=0
MOVL C00235 V=800.0 PL=0
MOVL C00236 V=800.0 PL=0
MOVL C00237 V=800.0 PL=0
MOVL C00238 V=800.0 PL=0
MOVL C00239 V=800.0 PL=0
MOVL C00240 V=800.0 PL=0
MOVL C00241 V=800.0 PL=0
MOVL C00242 V=800.0 PL=0
MOVL C00243 V=800.0 PL=0
MOVL C00244 V=800.0 PL=0
MOVL C00245 V=800.0 PL=0
MOVL C00246 V=800.0 PL=0
MOVL C00247 V=800.0 PL=0
MOVL C00248 V=800.0 PL=0
MOVL C00249 V=800.0 PL=0
MOVL C00250 V=800.0 PL=0
MOVL C00251 V=800.0 PL=0
MOVL C00252 V=800.0 PL=0
MOVL C00253 V=800.0 PL=0
MOVL C00254 V=800.0 PL=0
MOVL C00255 V=800.0 PL=0
MOVL C00256 V=800.0 PL=0
MOVL C00257 V=800.0 PL=0
MOVL C00258 V=800.0 PL=0
MOVL C00259 V=800.0 PL=0
MOVL C00260 V=800.0 PL=0
MOVL C00261 V=800.0 PL=0
MOVL C00262 V=800.0 PL=0
MOVL C00263 V=800.0 PL=0
MOVL C00264 V=800.0 PL=0
MOVL C00265 V=800.0 PL=0
MOVL C00266 V=800.0 PL=0
MOVL C00267 V=800.0 PL=0
MOVL C00268 V=800.0 PL=0
MOVL C00269 V=800.0 PL=0
MOVL C00270 V=800.0 PL=0
MOVL C00271 V=800.0 PL=0
MOVL C00272 V=800.0 PL=0
MOVL C00273 V=800.0 PL=0
MOVL C00274 V=800.0 PL=0
MOVL C00275 V=800.0 PL=0
MOVL C00276 V=800.0 PL=0
MOVL C00277 V=800.0 PL=0
MOVL C00278 V=800.0 PL=0
MOVL C00279 V=800.0 PL=0
MOVL C00280 V=800.0 PL=0
MOVL C00281 V=800.0 PL=0
MOVL C00282 V=800.0 PL=0
MOVL C00283 V=800.0 PL=0
MOVL C00284 V=800.0 PL=0
MOVL C00285 V=800.0 PL=0
MOVL C00286 V=800.0 PL=0
MOVL C00287 V=800.0 PL=0
MOVL C00288 V=800.0 PL=0
MOVL C00289 V=800.0 PL=0
MOVL C00290 V=800.0 PL=0
MOVL C00291 V=800.0 PL=0
MOVL C00292 V=800.0 PL=0
MOVL C00293 V=800.0 PL=0
MOVL C00294 V=800.0 PL=0
MOVL C00295 V=800.0 PL=0
MOVL C00296 V=800.0 PL=0
MOVL C00297 V=800.0 PL=0
MOVL C00298 V=800.0 PL=0
MOVL C00299 V=800.0 PL=0
MOVL C00300 V=800.0 PL=0
MOVL C00301 V=800.0 PL=0
MOVL C00302 V=800.0 PL=0
MOVL C00303 V=800.0 PL=0
MOVL C00304 V=800.0 PL=0
MOVL C00305 V=800.0 PL=0
MOVL C00306 V=800.0 PL=0
MOVL C00307 V=800.0 PL=0
MOVL C00308 V=800.0 PL=0
MOVL C00309 V=800.0 PL=0
MOVL C00310 V=800.0 PL=0
MOVL C00311 V=800.0 PL=0
MOVL C00312 V=800.0 PL=0
MOVL C00313 V=800.0 PL=0
MOVL C00314 V=800.0 PL=0
MOVL C00315 V=800.0 PL=0
MOVL C00316 V=800.0 PL=0
MOVL C00317 V=800.0 PL=0
MOVL C00318 V=800.0 PL=0
MOVL C00319 V=800.0 PL=0
MOVL C00320 V=800.0 PL=0
MOVL C00321 V=800.0 PL=0
MOVL C00322 V=800.0 PL=0
MOVL C00323 V=800.0 PL=0
MOVL C00324 V=800.0 PL=0
MOVL C00325 V=800.0 PL=0
MOVL C00326 V=800.0 PL=0
MOVL C00327 V=800.0 PL=0
MOVL C00328 V=800.0 PL=0
MOVL C00329 V=800.0 PL=0
MOVL C00330 V=800.0 PL=0
MOVL C00331 V=800.0 PL=0
MOVL C00332 V=800.0 PL=0
MOVL C00333 V=800.0 PL=0
MOVL C00334 V=800.0 PL=0
MOVL C00335 V=800.0 PL=0
MOVL C00336 V=800.0 PL=0
MOVL C00337 V=800.0 PL=0
MOVL C00338 V=800.0 PL=0
MOVL C00339 V=800.0 PL=0
MOVL C00340 V=800.0 PL=0
MOVL C00341 V=800.0 PL=0
MOVL C00342 V=800.0 PL=0
MOVL C00343 V=800.0 PL=0
MOVL C00344 V=800.0 PL=0
MOVL C00345 V=800.0 PL=0
MOVL C00346 V=800.0 PL=0
MOVL C00347 V=800.0 PL=0
MOVL C00348 V=800.0 PL=0
MOVL C00349 V=800.0 PL=0
MOVL C00350 V=800.0 PL=0
MOVL C00351 V=800.0 PL=0
MOVL C00352 V=800.0 PL=0
MOVL C00353 V=800.0 PL=0
MOVL C00354 V=800.0 PL=0
MOVL C00355 V=800.0 PL=0
MOVL C00356 V=800.0 PL=0
MOVL C00357 V=800.0 PL=0
MOVL C00358 V=800.0 PL=0
MOVL C00359 V=800.0 PL=0
MOVL C00360 V=800.0 PL=0
MOVL C00361 V=800.0 PL=0
MOVL C00362 V=800.0 PL=0
MOVL C00363 V=800.0 PL=0
MOVL C00364 V=800.0 PL=0
MOVL C00365 V=800.0 PL=0
MOVL C00366 V=800.0 PL=0
MOVL C00367 V=800.0 PL=0
MOVL C00368 V=800.0 PL=0
MOVL C00369 V=800.0 PL=0
MOVL C00370 V=800.0 PL=0
MOVL C00371 V=800.0 PL=0
MOVL C00372 V=800.0 PL=0
MOVL C00373 V=800.0 PL=0
MOVL C00374 V=800.0 PL=0
MOVL C00375 V=800.0 PL=0
MOVL C00376 V=800.0 PL=0
MOVL C00377 V=800.0 PL=0
MOVL C00378 V=800.0 PL=0
MOVL C00379 V=800.0 PL=0
MOVL C00380 V=800.0 PL=0
MOVL C00381 V=800.0 PL=0
MOVL C00382 V=800.0 PL=0
MOVL C00383 V=800.0 PL=0
MOVL C00384 V=800.0 PL=0
MOVL C00385 V=800.0 PL=0
MOVL C00386 V=800.0 PL=0
MOVL C00387 V=800.0 PL=0
MOVL C00388 V=800.0 PL=0
MOVL C00389 V=800.0 PL=0
MOVL C00390 V=800.0 PL=0
MOVL C00391 V=800.0 PL=0
MOVL C00392 V=800.0 PL=0
MOVL C00393 V=800.0 PL=0
MOVL C00394 V=800.0 PL=0
MOVL C00395 V=800.0 PL=0
MOVL C00396 V=800.0 PL=0
MOVL C00397 V=800.0 PL=0
MOVL C00398 V=800.0 PL=0
MOVL C00399 V=800.0 PL=0
MOVL C00400 V=800.0 PL=0
MOVL C00401 V=800.0 PL=0
MOVL C00402 V=800.0 PL=0
MOVL C00403 V=800.0 PL=0
MOVL C00404 V=800.0 PL=0
MOVL C00405 V=800.0 PL=0
MOVL C00406 V=800.0 PL=0
MOVL C00407 V=800.0 PL=0
MOVL C00408 V=800.0 PL=0
MOVL C00409 V=800.0 PL=0
MOVL C00410 V=800.0 PL=0
MOVL C00411 V=800.0 PL=0
MOVL C00412 V=800.0 PL=0
MOVL C00413 V=800.0 PL=0
MOVL C00414 V=800.0 PL=0
MOVL C00415 V=800.0 PL=0
MOVL C00416 V=800.0 PL=0
MOVL C00417 V=800.0 PL=0
MOVL C00418 V=800.0 PL=0
MOVL C00419 V=800.0 PL=0
MOVL C00420 V=800.0 PL=0
MOVL C00421 V=800.0 PL=0
MOVL C00422 V=800.0 PL=0
MOVL C00423 V=800.0 PL=0
MOVL C00424 V=800.0 PL=0
MOVL C00425 V=800.0 PL=0
MOVL C00426 V=800.0 PL=0
MOVL C00427 V=800.0 PL=0
MOVL C00428 V=800.0 PL=0
MOVL C00429 V=800.0 PL=0
MOVL C00430 V=800.0 PL=0
MOVL C00431 V=800.0 PL=0
MOVL C00432 V=800.0 PL=0
MOVL C00433 V=800.0 PL=0
MOVL C00434 V=800.0 PL=0
MOVL C00435 V=800.0 PL=0
MOVL C00436 V=800.0 PL=0
MOVL C00437 V=800.0 PL=0
MOVL C00438 V=800.0 PL=0
MOVL C00439 V=800.0 PL=0
MOVL C00440 V=800.0 PL=0
MOVL C00441 V=800.0 PL=0
MOVL C00442 V=800.0 PL=0
MOVL C00443 V=800.0 PL=0
MOVL C00444 V=800.0 PL=0
MOVL C00445 V=800.0 PL=0
MOVL C00446 V=800.0 PL=0
MOVL C00447 V=800.0 PL=0
MOVL C00448 V=800.0 PL=0
MOVL C00449 V=800.0 PL=0
MOVL C00450 V=800.0 PL=0
MOVL C00451 V=800.0 PL=0
MOVL C00452 V=800.0 PL=0
MOVL C00453 V=800.0 PL=0
MOVL C00454 V=800.0 PL=0
MOVL C00455 V=800.0 PL=0
MOVL C00456 V=800.0 PL=0
MOVL C00457 V=800.0 PL=0
MOVL C00458 V=800.0 PL=0
MOVL C00459 V=800.0 PL=0
MOVL C00460 V=800.0 PL=0
MOVL C00461 V=800.0 PL=0
MOVL C00462 V=800.0 PL=0
MOVL C00463 V=800.0 PL=0
MOVL C00464 V=800.0 PL=0
MOVL C00465 V=800.0 PL=0
MOVL C00466 V=800.0 PL=0
MOVL C00467 V=800.0 PL=0
MOVL C00468 V=800.0 PL=0
MOVL C00469 V=800.0 PL=0
MOVL C00470 V=800.0 PL=0
MOVL C00471 V=800.0 PL=0
MOVL C00472 V=800.0 PL=0
MOVL C00473 V=800.0 PL=0
MOVL C00474 V=800.0 PL=0
MOVL C00475 V=800.0 PL=0
MOVL C00476 V=800.0 PL=0
MOVL C00477 V=800.0 PL=0
MOVL C00478 V=800.0 PL=0
MOVL C00479 V=800.0 PL=0
MOVL C00480 V=800.0 PL=0
MOVL C00481 V=800.0 PL=0
MOVL C00482 V=800.0 PL=0
MOVL C00483 V=800.0 PL=0
MOVL C00484 V=800.0 PL=0
MOVL C00485 V=800.0 PL=0
MOVL C00486 V=800.0 PL=0
MOVL C00487 V=800.0 PL=0
MOVL C00488 V=800.0 PL=0
MOVL C00489 V=800.0 PL=0
MOVL C00490 V=800.0 PL=0
MOVL C00491 V=800.0 PL=0
MOVL C00492 V=800.0 PL=0
MOVL C00493 V=800.0 PL=0
MOVL C00494 V=800.0 PL=0
MOVL C00495 V=800.0 PL=0
MOVL C00496 V=800.0 PL=0
MOVL C00497 V=800.0 PL=0
MOVL C00498 V=800.0 PL=0
MOVL C00499 V=800.0 PL=0
MOVL C00500 V=800.0 PL=0
MOVL C00501 V=800.0 PL=0
MOVL C00502 V=800.0 PL=0
MOVL C00503 V=800.0 PL=0
MOVL C00504 V=800.0 PL=0
MOVL C00505 V=800.0 PL=0
MOVL C00506 V=800.0 PL=0
MOVL C00507 V=800.0 PL=0
MOVL C00508 V=800.0 PL=0
MOVL C00509 V=800.0 PL=0
MOVL C00510 V=800.0 PL=0
MOVL C00511 V=800.0 PL=0
MOVL C00512 V=800.0 PL=0
MOVL C00513 V=800.0 PL=0
MOVL C00514 V=800.0 PL=0
MOVL C00515 V=800.0 PL=0
MOVL C00516 V=800.0 PL=0
MOVL C00517 V=800.0 PL=0
MOVL C00518 V=800.0 PL=0
MOVL C00519 V=800.0 PL=0
MOVL C00520 V=800.0 PL=0
MOVL C00521 V=800.0 PL=0
MOVL C00522 V=800.0 PL=0
MOVL C00523 V=800.0 PL=0
MOVL C00524 V=800.0 PL=0
MOVL C00525 V=800.0 PL=0
MOVL C00526 V=800.0 PL=0
MOVL C00527 V=800.0 PL=0
MOVL C00528 V=800.0 PL=0
MOVL C00529 V=800.0 PL=0
MOVL C00530 V=800.0 PL=0
MOVL C00531 V=800.0 PL=0
MOVL C00532 V=800.0 PL=0
MOVL C00533 V=800.0 PL=0
MOVL C00534 V=800.0 PL=0
MOVL C00535 V=800.0 PL=0
MOVL C00536 V=800.0 PL=0
MOVL C00537 V=800.0 PL=0
MOVL C00538 V=800.0 PL=0
MOVL C00539 V=800.0 PL=0
MOVL C00540 V=800.0 PL=0
MOVL C00541 V=800.0 PL=0
MOVL C00542 V=800.0 PL=0
MOVL C00543 V=800.0 PL=0
MOVL C00544 V=800.0 PL=0
MOVL C00545 V=800.0 PL=0
MOVL C00546 V=800.0 PL=0
MOVL C00547 V=800.0 PL=0
MOVL C00548 V=800.0 PL=0
MOVL C00549 V=800.0 PL=0
MOVL C00550 V=800.0 PL=0
MOVL C00551 V=800.0 PL=0
MOVL C00552 V=800.0 PL=0
MOVL C00553 V=800.0 PL=0
MOVL C00554 V=800.0 PL=0
MOVL C00555 V=800.0 PL=0
MOVL C00556 V=800.0 PL=0
MOVL C00557 V=800.0 PL=0
MOVL C00558 V=800.0 PL=0
MOVL C00559 V=800.0 PL=0
MOVL C00560 V=800.0 PL=0
MOVL C00561 V=800.0 PL=0
MOVL C00562 V=800.0 PL=0
MOVL C00563 V=800.0 PL=0
MOVL C00564 V=800.0 PL=0
MOVL C00565 V=800.0 PL=0
MOVL C00566 V=800.0 PL=0
MOVL C00567 V=800.0 PL=0
MOVL C00568 V=800.0 PL=0
MOVL C00569 V=800.0 PL=0
MOVL C00570 V=800.0 PL=0
MOVL C00571 V=800.0 PL=0
MOVL C00572 V=800.0 PL=0
MOVL C00573 V=800.0 PL=0
MOVL C00574 V=800.0 PL=0
MOVL C00575 V=800.0 PL=0
MOVL C00576 V=800.0 PL=0
MOVL C00577 V=800.0 PL=0
MOVL C00578 V=800.0 PL=0
MOVL C00579 V=800.0 PL=0
MOVL C00580 V=800.0 PL=0
MOVL C00581 V=800.0 PL=0
MOVL C00582 V=800.0 PL=0
MOVL C00583 V=800.0 PL=0
MOVL C00584 V=800.0 PL=0
MOVL C00585 V=800.0 PL=0
MOVL C00586 V=800.0 PL=0
MOVL C00587 V=800.0 PL=0
MOVL C00588 V=800.0 PL=0
MOVL C00589 V=800.0 PL=0
MOVL C00590 V=800.0 PL=0
MOVL C00591 V=800.0 PL=0
MOVL C00592 V=800.0 PL=0
MOVL C00593 V=800.0 PL=0
MOVL C00594 V=800.0 PL=0
MOVL C00595 V=800.0 PL=0
MOVL C00596 V=800.0 PL=0
MOVL C00597 V=800.0 PL=0
MOVL C00598 V=800.0 PL=0
MOVL C00599 V=800.0 PL=0
MOVL C00600 V=800.0 PL=0
MOVL C00601 V=800.0 PL=0
MOVL C00602 V=800.0 PL=0
MOVL C00603 V=800.0 PL=0
MOVL C00604 V=800.0 PL=0
MOVL C00605 V=800.0 PL=0
MOVL C00606 V=800.0 PL=0
MOVL C00607 V=800.0 PL=0
MOVL C00608 V=800.0 PL=0
MOVL C00609 V=800.0 PL=0
MOVL C00610 V=800.0 PL=0
MOVL C00611 V=800.0 PL=0
MOVL C00612 V=800.0 PL=0
MOVL C00613 V=800.0 PL=0
MOVL C00614 V=800.0 PL=0
MOVL C00615 V=800.0 PL=0
MOVL C00616 V=800.0 PL=0
MOVL C00617 V=800.0 PL=0
MOVL C00618 V=800.0 PL=0
MOVL C00619 V=800.0 PL=0
MOVL C00620 V=800.0 PL=0
MOVL C00621 V=800.0 PL=0
MOVL C00622 V=800.0 PL=0
MOVL C00623 V=800.0 PL=0
MOVL C00624 V=800.0 PL=0
MOVL C00625 V=800.0 PL=0
MOVL C00626 V=800.0 PL=0
MOVL C00627 V=800.0 PL=0
MOVL C00628 V=800.0 PL=0
MOVL C00629 V=800.0 PL=0
MOVL C00630 V=800.0 PL=0
MOVL C00631 V=800.0 PL=0
MOVL C00632 V=800.0 PL=0
MOVL C00633 V=800.0 PL=0
MOVL C00634 V=800.0 PL=0
MOVL C00635 V=800.0 PL=0
MOVL C00636 V=800.0 PL=0
MOVL C00637 V=800.0 PL=0
MOVL C00638 V=800.0 PL=0
MOVL C00639 V=800.0 PL=0
MOVL C00640 V=800.0 PL=0
MOVL C00641 V=800.0 PL=0
MOVL C00642 V=800.0 PL=0
MOVL C00643 V=800.0 PL=0
MOVL C00644 V=800.0 PL=0
MOVL C00645 V=800.0 PL=0
MOVL C00646 V=800.0 PL=0
MOVL C00647 V=800.0 PL=0
MOVL C00648 V=800.0 PL=0
MOVL C00649 V=800.0 PL=0
MOVL C00650 V=800.0 PL=0
MOVL C00651 V=800.0 PL=0
MOVL C00652 V=800.0 PL=0
MOVL C00653 V=800.0 PL=0
MOVL C00654 V=800.0 PL=0
MOVL C00655 V=800.0 PL=0
MOVL C00656 V=800.0 PL=0
MOVL C00657 V=800.0 PL=0
MOVL C00658 V=800.0 PL=0
MOVL C00659 V=800.0 PL=0
MOVL C00660 V=800.0 PL=0
MOVL C00661 V=800.0 PL=0
MOVL C00662 V=800.0 PL=0
MOVL C00663 V=800.0 PL=0
MOVL C00664 V=800.0 PL=0
MOVL C00665 V=800.0 PL=0
MOVL C00666 V=800.0 PL=0
MOVL C00667 V=800.0 PL=0
MOVL C00668 V=800.0 PL=0
MOVL C00669 V=800.0 PL=0
MOVL C00670 V=800.0 PL=0
MOVL C00671 V=800.0 PL=0
MOVL C00672 V=800.0 PL=0
MOVL C00673 V=800.0 PL=0
MOVL C00674 V=800.0 PL=0
MOVL C00675 V=800.0 PL=0
MOVL C00676 V=800.0 PL=0
MOVL C00677 V=800.0 PL=0
MOVL C00678 V=800.0 PL=0
MOVL C00679 V=800.0 PL=0
MOVL C00680 V=800.0 PL=0
MOVL C00681 V=800.0 PL=0
MOVL C00682 V=800.0 PL=0
MOVL C00683 V=800.0 PL=0
MOVL C00684 V=800.0 PL=0
MOVL C00685 V=800.0 PL=0
MOVL C00686 V=800.0 PL=0
MOVL C00687 V=800.0 PL=0
MOVL C00688 V=800.0 PL=0
MOVL C00689 V=800.0 PL=0
MOVL C00690 V=800.0 PL=0
MOVL C00691 V=800.0 PL=0
MOVL C00692 V=800.0 PL=0
MOVL C00693 V=800.0 PL=0
MOVL C00694 V=800.0 PL=0
MOVL C00695 V=800.0 PL=0
MOVL C00696 V=800.0 PL=0
MOVL C00697 V=800.0 PL=0
MOVL C00698 V=800.0 PL=0
MOVL C00699 V=800.0 PL=0
MOVL C00700 V=800.0 PL=0
MOVL C00701 V=800.0 PL=0
MOVL C00702 V=800.0 PL=0
MOVL C00703 V=800.0 PL=0
MOVL C00704 V=800.0 PL=0
MOVL C00705 V=800.0 PL=0
MOVL C00706 V=800.0 PL=0
MOVL C00707 V=800.0 PL=0
MOVL C00708 V=800.0 PL=0
MOVL C00709 V=800.0 PL=0
MOVL C00710 V=800.0 PL=0
MOVL C00711 V=800.0 PL=0
MOVL C00712 V=800.0 PL=0
MOVL C00713 V=800.0 PL=0
MOVL C00714 V=800.0 PL=0
MOVL C00715 V=800.0 PL=0
MOVL C00716 V=800.0 PL=0
MOVL C00717 V=800.0 PL=0
MOVL C00718 V=800.0 PL=0
MOVL C00719 V=800.0 PL=0
MOVL C00720 V=800.0 PL=0
MOVL C00721 V=800.0 PL=0
MOVL C00722 V=800.0 PL=0
MOVL C00723 V=800.0 PL=0
MOVL C00724 V=800.0 PL=0
MOVL C00725 V=800.0 PL=0
MOVL C00726 V=800.0 PL=0
MOVL C00727 V=800.0 PL=0
MOVL C00728 V=800.0 PL=0
MOVL C00729 V=800.0 PL=0
MOVL C00730 V=800.0 PL=0
MOVL C00731 V=800.0 PL=0
MOVL C00732 V=800.0 PL=0
MOVL C00733 V=800.0 PL=0
MOVL C00734 V=800.0 PL=0
MOVL C00735 V=800.0 PL=0
MOVL C00736 V=800.0 PL=0
MOVL C00737 V=800.0 PL=0
MOVL C00738 V=800.0 PL=0
MOVL C00739 V=800.0 PL=0
MOVL C00740 V=800.0 PL=0
MOVL C00741 V=800.0 PL=0
MOVL C00742 V=800.0 PL=0
MOVL C00743 V=800.0 PL=0
MOVL C00744 V=800.0 PL=0
MOVL C00745 V=800.0 PL=0
MOVL C00746 V=800.0 PL=0
MOVL C00747 V=800.0 PL=0
MOVL C00748 V=800.0 PL=0
MOVL C00749 V=800.0 PL=0
MOVL C00750 V=800.0 PL=0
MOVL C00751 V=800.0 PL=0
MOVL C00752 V=800.0 PL=0
MOVL C00753 V=800.0 PL=0
MOVL C00754 V=800.0 PL=0
MOVL C00755 V=800.0 PL=0
MOVL C00756 V=800.0 PL=0
MOVL C00757 V=800.0 PL=0
MOVL C00758 V=800.0 PL=0
MOVL C00759 V=800.0 PL=0
MOVL C00760 V=800.0 PL=0
MOVL C00761 V=800.0 PL=0
MOVL C00762 V=800.0 PL=0
MOVL C00763 V=800.0 PL=0
MOVL C00764 V=800.0 PL=0
MOVL C00765 V=800.0 PL=0
MOVL C00766 V=800.0 PL=0
MOVL C00767 V=800.0 PL=0
MOVL C00768 V=800.0 PL=0
MOVL C00769 V=800.0 PL=0
MOVL C00770 V=800.0 PL=0
MOVL C00771 V=800.0 PL=0
MOVL C00772 V=800.0 PL=0
MOVL C00773 V=800.0 PL=0
MOVL C00774 V=800.0 PL=0
MOVL C00775 V=800.0 PL=0
MOVL C00776 V=800.0 PL=0
MOVL C00777 V=800.0 PL=0
MOVL C00778 V=800.0 PL=0
MOVL C00779 V=800.0 PL=0
MOVL C00780 V=800.0 PL=0
MOVL C00781 V=800.0 PL=0
MOVL C00782 V=800.0 PL=0
MOVL C00783 V=800.0 PL=0
MOVL C00784 V=800.0 PL=0
MOVL C00785 V=800.0 PL=0
MOVL C00786 V=800.0 PL=0
MOVL C00787 V=800.0 PL=0
MOVL C00788 V=800.0 PL=0
MOVL C00789 V=800.0 PL=0
MOVL C00790 V=800.0 PL=0
MOVL C00791 V=800.0 PL=0
MOVL C00792 V=800.0 PL=0
MOVL C00793 V=800.0 PL=0
MOVL C00794 V=800.0 PL=0
MOVL C00795 V=800.0 PL=0
MOVL C00796 V=800.0 PL=0
MOVL C00797 V=800.0 PL=0
MOVL C00798 V=800.0 PL=0
MOVL C00799 V=800.0 PL=0
MOVL C00800 V=800.0 PL=0
MOVL C00801 V=800.0 PL=0
MOVL C00802 V=800.0 PL=0
MOVL C00803 V=800.0 PL=0
MOVL C00804 V=800.0 PL=0
MOVL C00805 V=800.0 PL=0
MOVL C00806 V=800.0 PL=0
MOVL C00807 V=800.0 PL=0
MOVL C00808 V=800.0 PL=0
MOVL C00809 V=800.0 PL=0
MOVL C00810 V=800.0 PL=0
MOVL C00811 V=800.0 PL=0
MOVL C00812 V=800.0 PL=0
MOVL C00813 V=800.0 PL=0
MOVL C00814 V=800.0 PL=0
MOVL C00815 V=800.0 PL=0
MOVL C00816 V=800.0 PL=0
MOVL C00817 V=800.0 PL=0
MOVL C00818 V=800.0 PL=0
MOVL C00819 V=800.0 PL=0
MOVL C00820 V=800.0 PL=0
MOVL C00821 V=800.0 PL=0
MOVL C00822 V=800.0 PL=0
MOVL C00823 V=800.0 PL=0
MOVL C00824 V=800.0 PL=0
MOVL C00825 V=800.0 PL=0
MOVL C00826 V=800.0 PL=0
MOVL C00827 V=800.0 PL=0
MOVL C00828 V=800.0 PL=0
MOVL C00829 V=800.0 PL=0
MOVL C00830 V=800.0 PL=0
MOVL C00831 V=800.0 PL=0
MOVL C00832 V=800.0 PL=0
MOVL C00833 V=800.0 PL=0
MOVL C00834 V=800.0 PL=0
MOVL C00835 V=800.0 PL=0
MOVL C00836 V=800.0 PL=0
MOVL C00837 V=800.0 PL=0
MOVL C00838 V=800.0 PL=0
MOVL C00839 V=800.0 PL=0
MOVL C00840 V=800.0 PL=0
MOVL C00841 V=800.0 PL=0
MOVL C00842 V=800.0 PL=0
MOVL C00843 V=800.0 PL=0
MOVL C00844 V=800.0 PL=0
MOVL C00845 V=800.0 PL=0
MOVL C00846 V=800.0 PL=0
MOVL C00847 V=800.0 PL=0
MOVL C00848 V=800.0 PL=0
MOVL C00849 V=800.0 PL=0
MOVL C00850 V=800.0 PL=0
MOVL C00851 V=800.0 PL=0
MOVL C00852 V=800.0 PL=0
MOVL C00853 V=800.0 PL=0
MOVL C00854 V=800.0 PL=0
MOVL C00855 V=800.0 PL=0
MOVL C00856 V=800.0 PL=0
MOVL C00857 V=800.0 PL=0
MOVL C00858 V=800.0 PL=0
MOVL C00859 V=800.0 PL=0
MOVL C00860 V=800.0 PL=0
MOVL C00861 V=800.0 PL=0
MOVL C00862 V=800.0 PL=0
MOVL C00863 V=800.0 PL=0
MOVL C00864 V=800.0 PL=0
MOVL C00865 V=800.0 PL=0
MOVL C00866 V=800.0 PL=0
MOVL C00867 V=800.0 PL=0
MOVL C00868 V=800.0 PL=0
MOVL C00869 V=800.0 PL=0
MOVL C00870 V=800.0 PL=0
MOVL C00871 V=800.0 PL=0
MOVL C00872 V=800.0 PL=0
MOVL C00873 V=800.0 PL=0
MOVL C00874 V=800.0 PL=0
MOVL C00875 V=800.0 PL=0
MOVL C00876 V=800.0 PL=0
MOVL C00877 V=800.0 PL=0
MOVL C00878 V=800.0 PL=0
MOVL C00879 V=800.0 PL=0
MOVL C00880 V=800.0 PL=0
MOVL C00881 V=800.0 PL=0
MOVL C00882 V=800.0 PL=0
MOVL C00883 V=800.0 PL=0
MOVL C00884 V=800.0 PL=0
MOVL C00885 V=800.0 PL=0
MOVL C00886 V=800.0 PL=0
MOVL C00887 V=800.0 PL=0
MOVL C00888 V=800.0 PL=0
MOVL C00889 V=800.0 PL=0
MOVL C00890 V=800.0 PL=0
MOVL C00891 V=800.0 PL=0
MOVL C00892 V=800.0 PL=0
MOVL C00893 V=800.0 PL=0
MOVL C00894 V=800.0 PL=0
MOVL C00895 V=800.0 PL=0
MOVL C00896 V=800.0 PL=0
MOVL C00897 V=800.0 PL=0
MOVL C00898 V=800.0 PL=0
MOVL C00899 V=800.0 PL=0
MOVL C00900 V=800.0 PL=0
MOVL C00901 V=800.0 PL=0
MOVL C00902 V=800.0 PL=0
MOVL C00903 V=800.0 PL=0
MOVL C00904 V=800.0 PL=0
MOVL C00905 V=800.0 PL=0
MOVL C00906 V=800.0 PL=0
MOVL C00907 V=800.0 PL=0
MOVL C00908 V=800.0 PL=0
MOVL C00909 V=800.0 PL=0
MOVL C00910 V=800.0 PL=0
MOVL C00911 V=800.0 PL=0
MOVL C00912 V=800.0 PL=0
MOVL C00913 V=800.0 PL=0
MOVL C00914 V=800.0 PL=0
MOVL C00915 V=800.0 PL=0
MOVL C00916 V=800.0 PL=0
MOVL C00917 V=800.0 PL=0
MOVL C00918 V=800.0 PL=0
MOVL C00919 V=800.0 PL=0
MOVL C00920 V=800.0 PL=0
MOVL C00921 V=800.0 PL=0
MOVL C00922 V=800.0 PL=0
MOVL C00923 V=800.0 PL=0
MOVL C00924 V=800.0 PL=0
MOVL C00925 V=800.0 PL=0
MOVL C00926 V=800.0 PL=0
MOVL C00927 V=800.0 PL=0
MOVL C00928 V=800.0 PL=0
MOVL C00929 V=800.0 PL=0
MOVL C00930 V=800.0 PL=0
MOVL C00931 V=800.0 PL=0
MOVL C00932 V=800.0 PL=0
MOVL C00933 V=800.0 PL=0
MOVL C00934 V=800.0 PL=0
MOVL C00935 V=800.0 PL=0
MOVL C00936 V=800.0 PL=0
MOVL C00937 V=800.0 PL=0
MOVL C00938 V=800.0 PL=0
MOVL C00939 V=800.0 PL=0
MOVL C00940 V=800.0 PL=0
MOVL C00941 V=800.0 PL=0
MOVL C00942 V=800.0 PL=0
MOVL C00943 V=800.0 PL=0
MOVL C00944 V=800.0 PL=0
MOVL C00945 V=800.0 PL=0
MOVL C00946 V=800.0 PL=0
MOVL C00947 V=800.0 PL=0
MOVL C00948 V=800.0 PL=0
MOVL C00949 V=800.0 PL=0
MOVL C00950 V=800.0 PL=0
MOVL C00951 V=800.0 PL=0
MOVL C00952 V=800.0 PL=0
MOVL C00953 V=800.0 PL=0
MOVL C00954 V=800.0 PL=0
MOVL C00955 V=800.0 PL=0
MOVL C00956 V=800.0 PL=0
MOVL C00957 V=800.0 PL=0
MOVL C00958 V=800.0 PL=0
MOVL C00959 V=800.0 PL=0
MOVL C00960 V=800.0 PL=0
MOVL C00961 V=800.0 PL=0
MOVL C00962 V=800.0 PL=0
MOVL C00963 V=800.0 PL=0
MOVL C00964 V=800.0 PL=0
MOVL C00965 V=800.0 PL=0
MOVL C00966 V=800.0 PL=0
MOVL C00967 V=800.0 PL=0
MOVL C00968 V=800.0 PL=0
MOVL C00969 V=800.0 PL=0
MOVL C00970 V=800.0 PL=0
MOVL C00971 V=800.0 PL=0
MOVL C00972 V=800.0 PL=0
MOVL C00973 V=800.0 PL=0
MOVL C00974 V=800.0 PL=0
MOVL C00975 V=800.0 PL=0
MOVL C00976 V=800.0 PL=0
MOVL C00977 V=800.0 PL=0
MOVL C00978 V=800.0 PL=0
MOVL C00979 V=800.0 PL=0
MOVL C00980 V=800.0 PL=0
MOVL C00981 V=800.0 PL=0
MOVL C00982 V=800.0 PL=0
MOVL C00983 V=800.0 PL=0
MOVL C00984 V=800.0 PL=0
MOVL C00985 V=800.0 PL=0
MOVL C00986 V=800.0 PL=0
MOVL C00987 V=800.0 PL=0
MOVL C00988 V=800.0 PL=0
MOVL C00989 V=800.0 PL=0
MOVL C00990 V=800.0 PL=0
MOVL C00991 V=800.0 PL=0
MOVL C00992 V=800.0 PL=0
MOVL C00993 V=800.0 PL=0
MOVL C00994 V=800.0 PL=0
MOVL C00995 V=800.0 PL=0
MOVL C00996 V=800.0 PL=0
MOVL C00997 V=800.0 PL=0
MOVL C00998 V=800.0 PL=0
MOVL C00999 V=800.0 PL=0
MOVL C01000 V=800.0 PL=0
MOVL C01001 V=800.0 PL=0
MOVL C01002 V=800.0 PL=0
MOVL C01003 V=800.0 PL=0
MOVL C01004 V=800.0 PL=0
MOVL C01005 V=800.0 PL=0
MOVL C01006 V=800.0 PL=0
MOVL C01007 V=800.0 PL=0
MOVL C01008 V=800.0 PL=0
MOVL C01009 V=800.0 PL=0
MOVL C01010 V=800.0 PL=0
MOVL C01011 V=800.0 PL=0
MOVL C01012 V=800.0 PL=0
MOVL C01013 V=800.0 PL=0
MOVL C01014 V=800.0 PL=0
MOVL C01015 V=800.0 PL=0
MOVL C01016 V=800.0 PL=0
MOVL C01017 V=800.0 PL=0
MOVL C01018 V=800.0 PL=0
MOVL C01019 V=800.0 PL=0
MOVL C01020 V=800.0 PL=0
MOVL C01021 V=800.0 PL=0
MOVL C01022 V=800.0 PL=0
MOVL C01023 V=800.0 PL=0
MOVL C01024 V=800.0 PL=0
MOVL C01025 V=800.0 PL=0
MOVL C01026 V=800.0 PL=0
MOVL C01027 V=800.0 PL=0
MOVL C01028 V=800.0 PL=0
MOVL C01029 V=800.0 PL=0
MOVL C01030 V=800.0 PL=0
MOVL C01031 V=800.0 PL=0
MOVL C01032 V=800.0 PL=0
MOVL C01033 V=800.0 PL=0
MOVL C01034 V=800.0 PL=0
MOVL C01035 V=800.0 PL=0
MOVL C01036 V=800.0 PL=0
MOVL C01037 V=800.0 PL=0
MOVL C01038 V=800.0 PL=0
MOVL C01039 V=800.0 PL=0
MOVL C01040 V=800.0 PL=0
MOVL C01041 V=800.0 PL=0
MOVL C01042 V=800.0 PL=0
MOVL C01043 V=800.0 PL=0
MOVL C01044 V=800.0 PL=0
MOVL C01045 V=800.0 PL=0
MOVL C01046 V=800.0 PL=0
MOVL C01047 V=800.0 PL=0
MOVL C01048 V=800.0 PL=0
MOVL C01049 V=800.0 PL=0
MOVL C01050 V=800.0 PL=0
MOVL C01051 V=800.0 PL=0
MOVL C01052 V=800.0 PL=0
MOVL C01053 V=800.0 PL=0
MOVL C01054 V=800.0 PL=0
MOVL C01055 V=800.0 PL=0
MOVL C01056 V=800.0 PL=0
MOVL C01057 V=800.0 PL=0
MOVL C01058 V=800.0 PL=0
MOVL C01059 V=800.0 PL=0
MOVL C01060 V=800.0 PL=0
MOVL C01061 V=800.0 PL=0
MOVL C01062 V=800.0 PL=0
MOVL C01063 V=800.0 PL=0
MOVL C01064 V=800.0 PL=0
MOVL C01065 V=800.0 PL=0
MOVL C01066 V=800.0 PL=0
MOVL C01067 V=800.0 PL=0
MOVL C01068 V=800.0 PL=0
MOVL C01069 V=800.0 PL=0
MOVL C01070 V=800.0 PL=0
MOVL C01071 V=800.0 PL=0
MOVL C01072 V=800.0 PL=0
MOVL C01073 V=800.0 PL=0
MOVL C01074 V=800.0 PL=0
MOVL C01075 V=800.0 PL=0
MOVL C01076 V=800.0 PL=0
MOVL C01077 V=800.0 PL=0
MOVL C01078 V=800.0 PL=0
MOVL C01079 V=800.0 PL=0
MOVL C01080 V=800.0 PL=0
MOVL C01081 V=800.0 PL=0
MOVL C01082 V=800.0 PL=0
MOVL C01083 V=800.0 PL=0
MOVL C01084 V=800.0 PL=0
MOVL C01085 V=800.0 PL=0
MOVL C01086 V=800.0 PL=0
MOVL C01087 V=800.0 PL=0
MOVL C01088 V=800.0 PL=0
MOVL C01089 V=800.0 PL=0
MOVL C01090 V=800.0 PL=0
MOVL C01091 V=800.0 PL=0
MOVL C01092 V=800.0 PL=0
MOVL C01093 V=800.0 PL=0
MOVL C01094 V=800.0 PL=0
MOVL C01095 V=800.0 PL=0
MOVL C01096 V=800.0 PL=0
MOVL C01097 V=800.0 PL=0
MOVL C01098 V=800.0 PL=0
MOVL C01099 V=800.0 PL=0
MOVL C01100 V=800.0 PL=0
MOVL C01101 V=800.0 PL=0
MOVL C01102 V=800.0 PL=0
MOVL C01103 V=800.0 PL=0
MOVL C01104 V=800.0 PL=0
MOVL C01105 V=800.0 PL=0
MOVL C01106 V=800.0 PL=0
MOVL C01107 V=800.0 PL=0
MOVL C01108 V=800.0 PL=0
MOVL C01109 V=800.0 PL=0
MOVL C01110 V=800.0 PL=0
MOVL C01111 V=800.0 PL=0
MOVL C01112 V=800.0 PL=0
MOVL C01113 V=800.0 PL=0
MOVL C01114 V=800.0 PL=0
MOVL C01115 V=800.0 PL=0
MOVL C01116 V=800.0 PL=0
MOVL C01117 V=800.0 PL=0
MOVL C01118 V=800.0 PL=0
MOVL C01119 V=800.0 PL=0
MOVL C01120 V=800.0 PL=0
MOVL C01121 V=800.0 PL=0
MOVL C01122 V=800.0 PL=0
MOVL C01123 V=800.0 PL=0
MOVL C01124 V=800.0 PL=0
MOVL C01125 V=800.0 PL=0
MOVL C01126 V=800.0 PL=0
MOVL C01127 V=800.0 PL=0
MOVL C01128 V=800.0 PL=0
MOVL C01129 V=800.0 PL=0
MOVL C01130 V=800.0 PL=0
MOVL C01131 V=800.0 PL=0
MOVL C01132 V=800.0 PL=0
MOVL C01133 V=800.0 PL=0
MOVL C01134 V=800.0 PL=0
MOVL C01135 V=800.0 PL=0
MOVL C01136 V=800.0 PL=0
MOVL C01137 V=800.0 PL=0
MOVL C01138 V=800.0 PL=0
MOVL C01139 V=800.0 PL=0
MOVL C01140 V=800.0 PL=0
MOVL C01141 V=800.0 PL=0
MOVL C01142 V=800.0 PL=0
MOVL C01143 V=800.0 PL=0
MOVL C01144 V=800.0 PL=0
MOVL C01145 V=800.0 PL=0
MOVL C01146 V=800.0 PL=0
MOVL C01147 V=800.0 PL=0
MOVL C01148 V=800.0 PL=0
MOVL C01149 V=800.0 PL=0
MOVL C01150 V=800.0 PL=0
MOVL C01151 V=800.0 PL=0
MOVL C01152 V=800.0 PL=0
MOVL C01153 V=800.0 PL=0
MOVL C01154 V=800.0 PL=0
MOVL C01155 V=800.0 PL=0
MOVL C01156 V=800.0 PL=0
MOVL C01157 V=800.0 PL=0
MOVL C01158 V=800.0 PL=0
MOVL C01159 V=800.0 PL=0
MOVL C01160 V=800.0 PL=0
MOVL C01161 V=800.0 PL=0
MOVL C01162 V=800.0 PL=0
MOVL C01163 V=800.0 PL=0
MOVL C01164 V=800.0 PL=0
MOVL C01165 V=800.0 PL=0
MOVL C01166 V=800.0 PL=0
MOVL C01167 V=800.0 PL=0
MOVL C01168 V=800.0 PL=0
MOVL C01169 V=800.0 PL=0
MOVL C01170 V=800.0 PL=0
MOVL C01171 V=800.0 PL=0
MOVL C01172 V=800.0 PL=0
MOVL C01173 V=800.0 PL=0
MOVL C01174 V=800.0 PL=0
MOVL C01175 V=800.0 PL=0
MOVL C01176 V=800.0 PL=0
MOVL C01177 V=800.0 PL=0
MOVL C01178 V=800.0 PL=0
MOVL C01179 V=800.0 PL=0
MOVL C01180 V=800.0 PL=0
MOVL C01181 V=800.0 PL=0
MOVL C01182 V=800.0 PL=0
MOVL C01183 V=800.0 PL=0
MOVL C01184 V=800.0 PL=0
MOVL C01185 V=800.0 PL=0
MOVL C01186 V=800.0 PL=0
MOVL C01187 V=800.0 PL=0
MOVL C01188 V=800.0 PL=0
MOVL C01189 V=800.0 PL=0
MOVL C01190 V=800.0 PL=0
MOVL C01191 V=800.0 PL=0
MOVL C01192 V=800.0 PL=0
MOVL C01193 V=800.0 PL=0
MOVL C01194 V=800.0 PL=0
MOVL C01195 V=800.0 PL=0
MOVL C01196 V=800.0 PL=0
MOVL C01197 V=800.0 PL=0
MOVL C01198 V=800.0 PL=0
MOVL C01199 V=800.0 PL=0
MOVL C01200 V=800.0 PL=0
MOVL C01201 V=800.0 PL=0
MOVL C01202 V=800.0 PL=0
MOVL C01203 V=800.0 PL=0
MOVL C01204 V=800.0 PL=0
MOVL C01205 V=800.0 PL=0
MOVL C01206 V=800.0 PL=0
MOVL C01207 V=800.0 PL=0
MOVL C01208 V=800.0 PL=0
MOVL C01209 V=800.0 PL=0
MOVL C01210 V=800.0 PL=0
MOVL C01211 V=800.0 PL=0
MOVL C01212 V=800.0 PL=0
MOVL C01213 V=800.0 PL=0
MOVL C01214 V=800.0 PL=0
MOVL C01215 V=800.0 PL=0
MOVL C01216 V=800.0 PL=0
MOVL C01217 V=800.0 PL=0
MOVL C01218 V=800.0 PL=0
MOVL C01219 V=800.0 PL=0
MOVL C01220 V=800.0 PL=0
MOVL C01221 V=800.0 PL=0
MOVL C01222 V=800.0 PL=0
MOVL C01223 V=800.0 PL=0
MOVL C01224 V=800.0 PL=0
MOVL C01225 V=800.0 PL=0
MOVL C01226 V=800.0 PL=0
MOVL C01227 V=800.0 PL=0
MOVL C01228 V=800.0 PL=0
MOVL C01229 V=800.0 PL=0
MOVL C01230 V=800.0 PL=0
MOVL C01231 V=800.0 PL=0
MOVL C01232 V=800.0 PL=0
MOVL C01233 V=800.0 PL=0
MOVL C01234 V=800.0 PL=0
MOVL C01235 V=800.0 PL=0
MOVL C01236 V=800.0 PL=0
MOVL C01237 V=800.0 PL=0
MOVL C01238 V=800.0 PL=0
MOVL C01239 V=800.0 PL=0
MOVL C01240 V=800.0 PL=0
MOVL C01241 V=800.0 PL=0
MOVL C01242 V=800.0 PL=0
MOVL C01243 V=800.0 PL=0
MOVL C01244 V=800.0 PL=0
MOVL C01245 V=800.0 PL=0
MOVL C01246 V=800.0 PL=0
MOVL C01247 V=800.0 PL=0
MOVL C01248 V=800.0 PL=0
MOVL C01249 V=800.0 PL=0
MOVL C01250 V=800.0 PL=0
MOVL C01251 V=800.0 PL=0
MOVL C01252 V=800.0 PL=0
MOVL C01253 V=800.0 PL=0
MOVL C01254 V=800.0 PL=0
MOVL C01255 V=800.0 PL=0
MOVL C01256 V=800.0 PL=0
MOVL C01257 V=800.0 PL=0
MOVL C01258 V=800.0 PL=0
MOVL C01259 V=800.0 PL=0
MOVL C01260 V=800.0 PL=0
MOVL C01261 V=800.0 PL=0
MOVL C01262 V=800.0 PL=0
MOVL C01263 V=800.0 PL=0
MOVL C01264 V=800.0 PL=0
MOVL C01265 V=800.0 PL=0
MOVL C01266 V=800.0 PL=0
MOVL C01267 V=800.0 PL=0
MOVL C01268 V=800.0 PL=0
MOVL C01269 V=800.0 PL=0
MOVL C01270 V=800.0 PL=0
MOVL C01271 V=800.0 PL=0
MOVL C01272 V=800.0 PL=0
MOVL C01273 V=800.0 PL=0
MOVL C01274 V=800.0 PL=0
MOVL C01275 V=800.0 PL=0
MOVL C01276 V=800.0 PL=0
MOVL C01277 V=800.0 PL=0
MOVL C01278 V=800.0 PL=0
MOVL C01279 V=800.0 PL=0
MOVL C01280 V=800.0 PL=0
MOVL C01281 V=800.0 PL=0
MOVL C01282 V=800.0 PL=0
MOVL C01283 V=800.0 PL=0
MOVL C01284 V=800.0 PL=0
MOVL C01285 V=800.0 PL=0
MOVL C01286 V=800.0 PL=0
MOVL C01287 V=800.0 PL=0
MOVL C01288 V=800.0 PL=0
MOVL C01289 V=800.0 PL=0
MOVL C01290 V=800.0 PL=0
MOVL C01291 V=800.0 PL=0
MOVL C01292 V=800.0 PL=0
MOVL C01293 V=800.0 PL=0
MOVL C01294 V=800.0 PL=0
MOVL C01295 V=800.0 PL=0
MOVL C01296 V=800.0 PL=0
MOVL C01297 V=800.0 PL=0
MOVL C01298 V=800.0 PL=0
MOVL C01299 V=800.0 PL=0
MOVL C01300 V=800.0 PL=0
MOVL C01301 V=800.0 PL=0
MOVL C01302 V=800.0 PL=0
MOVL C01303 V=800.0 PL=0
MOVL C01304 V=800.0 PL=0
MOVL C01305 V=800.0 PL=0
MOVL C01306 V=800.0 PL=0
MOVL C01307 V=800.0 PL=0
MOVL C01308 V=800.0 PL=0
MOVL C01309 V=800.0 PL=0
MOVL C01310 V=800.0 PL=0
MOVL C01311 V=800.0 PL=0
MOVL C01312 V=800.0 PL=0
MOVL C01313 V=800.0 PL=0
MOVL C01314 V=800.0 PL=0
MOVL C01315 V=800.0 PL=0
MOVL C01316 V=800.0 PL=0
MOVL C01317 V=800.0 PL=0
MOVL C01318 V=800.0 PL=0
MOVL C01319 V=800.0 PL=0
MOVL C01320 V=800.0 PL=0
MOVL C01321 V=800.0 PL=0
MOVL C01322 V=800.0 PL=0
MOVL C01323 V=800.0 PL=0
MOVL C01324 V=800.0 PL=0
MOVL C01325 V=800.0 PL=0
MOVL C01326 V=800.0 PL=0
MOVL C01327 V=800.0 PL=0
MOVL C01328 V=800.0 PL=0
MOVL C01329 V=800.0 PL=0
MOVL C01330 V=800.0 PL=0
MOVL C01331 V=800.0 PL=0
MOVL C01332 V=800.0 PL=0
MOVL C01333 V=800.0 PL=0
MOVL C01334 V=800.0 PL=0
MOVL C01335 V=800.0 PL=0
MOVL C01336 V=800.0 PL=0
MOVL C01337 V=800.0 PL=0
MOVL C01338 V=800.0 PL=0
MOVL C01339 V=800.0 PL=0
MOVL C01340 V=800.0 PL=0
MOVL C01341 V=800.0 PL=0
MOVL C01342 V=800.0 PL=0
MOVL C01343 V=800.0 PL=0
MOVL C01344 V=800.0 PL=0
MOVL C01345 V=800.0 PL=0
MOVL C01346 V=800.0 PL=0
MOVL C01347 V=800.0 PL=0
MOVL C01348 V=800.0 PL=0
MOVL C01349 V=800.0 PL=0
MOVL C01350 V=800.0 PL=0
MOVL C01351 V=800.0 PL=0
MOVL C01352 V=800.0 PL=0
MOVL C01353 V=800.0 PL=0
MOVL C01354 V=800.0 PL=0
MOVL C01355 V=800.0 PL=0
MOVL C01356 V=800.0 PL=0
MOVL C01357 V=800.0 PL=0
MOVL C01358 V=800.0 PL=0
MOVL C01359 V=800.0 PL=0
MOVL C01360 V=800.0 PL=0
MOVL C01361 V=800.0 PL=0
MOVL C01362 V=800.0 PL=0
MOVL C01363 V=800.0 PL=0
MOVL C01364 V=800.0 PL=0
MOVL C01365 V=800.0 PL=0
MOVL C01366 V=800.0 PL=0
MOVL C01367 V=800.0 PL=0
MOVL C01368 V=800.0 PL=0
MOVL C01369 V=800.0 PL=0
MOVL C01370 V=800.0 PL=0
MOVL C01371 V=800.0 PL=0
MOVL C01372 V=800.0 PL=0
MOVL C01373 V=800.0 PL=0
MOVL C01374 V=800.0 PL=0
MOVL C01375 V=800.0 PL=0
MOVL C01376 V=800.0 PL=0
MOVL C01377 V=800.0 PL=0
MOVL C01378 V=800.0 PL=0
MOVL C01379 V=800.0 PL=0
MOVL C01380 V=800.0 PL=0
MOVL C01381 V=800.0 PL=0
MOVL C01382 V=800.0 PL=0
MOVL C01383 V=800.0 PL=0
MOVL C01384 V=800.0 PL=0
MOVL C01385 V=800.0 PL=0
MOVL C01386 V=800.0 PL=0
MOVL C01387 V=800.0 PL=0
MOVL C01388 V=800.0 PL=0
MOVL C01389 V=800.0 PL=0
MOVL C01390 V=800.0 PL=0
MOVL C01391 V=800.0 PL=0
MOVL C01392 V=800.0 PL=0
MOVL C01393 V=800.0 PL=0
MOVL C01394 V=800.0 PL=0
MOVL C01395 V=800.0 PL=0
MOVL C01396 V=800.0 PL=0
MOVL C01397 V=800.0 PL=0
MOVL C01398 V=800.0 PL=0
MOVL C01399 V=800.0 PL=0
MOVL C01400 V=800.0 PL=0
MOVL C01401 V=800.0 PL=0
MOVL C01402 V=800.0 PL=0
MOVL C01403 V=800.0 PL=0
MOVL C01404 V=800.0 PL=0
MOVL C01405 V=800.0 PL=0
MOVL C01406 V=800.0 PL=0
MOVL C01407 V=800.0 PL=0
MOVL C01408 V=800.0 PL=0
MOVL C01409 V=800.0 PL=0
MOVL C01410 V=800.0 PL=0
MOVL C01411 V=800.0 PL=0
MOVL C01412 V=800.0 PL=0
MOVL C01413 V=800.0 PL=0
MOVL C01414 V=800.0 PL=0
MOVL C01415 V=800.0 PL=0
MOVL C01416 V=800.0 PL=0
MOVL C01417 V=800.0 PL=0
MOVL C01418 V=800.0 PL=0
MOVL C01419 V=800.0 PL=0
MOVL C01420 V=800.0 PL=0
MOVL C01421 V=800.0 PL=0
MOVL C01422 V=800.0 PL=0
MOVL C01423 V=800.0 PL=0
MOVL C01424 V=800.0 PL=0
MOVL C01425 V=800.0 PL=0
MOVL C01426 V=800.0 PL=0
MOVL C01427 V=800.0 PL=0
MOVL C01428 V=800.0 PL=0
MOVL C01429 V=800.0 PL=0
MOVL C01430 V=800.0 PL=0
MOVL C01431 V=800.0 PL=0
MOVL C01432 V=800.0 PL=0
MOVL C01433 V=800.0 PL=0
MOVL C01434 V=800.0 PL=0
MOVL C01435 V=800.0 PL=0
MOVL C01436 V=800.0 PL=0
MOVL C01437 V=800.0 PL=0
MOVL C01438 V=800.0 PL=0
MOVL C01439 V=800.0 PL=0
MOVL C01440 V=800.0 PL=0
MOVL C01441 V=800.0 PL=0
MOVL C01442 V=800.0 PL=0
MOVL C01443 V=800.0 PL=0
MOVL C01444 V=800.0 PL=0
MOVL C01445 V=800.0 PL=0
MOVL C01446 V=800.0 PL=0
MOVL C01447 V=800.0 PL=0
MOVL C01448 V=800.0 PL=0
MOVL C01449 V=800.0 PL=0
MOVL C01450 V=800.0 PL=0
MOVL C01451 V=800.0 PL=0
MOVL C01452 V=800.0 PL=0
MOVL C01453 V=800.0 PL=0
MOVL C01454 V=800.0 PL=0
MOVL C01455 V=800.0 PL=0
MOVL C01456 V=800.0 PL=0
MOVL C01457 V=800.0 PL=0
MOVL C01458 V=800.0 PL=0
MOVL C01459 V=800.0 PL=0
MOVL C01460 V=800.0 PL=0
MOVL C01461 V=800.0 PL=0
MOVL C01462 V=800.0 PL=0
MOVL C01463 V=800.0 PL=0
MOVL C01464 V=800.0 PL=0
MOVL C01465 V=800.0 PL=0
MOVL C01466 V=800.0 PL=0
MOVL C01467 V=800.0 PL=0
MOVL C01468 V=800.0 PL=0
MOVL C01469 V=800.0 PL=0
MOVL C01470 V=800.0 PL=0
MOVL C01471 V=800.0 PL=0
MOVL C01472 V=800.0 PL=0
MOVL C01473 V=800.0 PL=0
MOVL C01474 V=800.0 PL=0
MOVL C01475 V=800.0 PL=0
MOVL C01476 V=800.0 PL=0
MOVL C01477 V=800.0 PL=0
MOVL C01478 V=800.0 PL=0
MOVL C01479 V=800.0 PL=0
MOVL C01480 V=800.0 PL=0
MOVL C01481 V=800.0 PL=0
MOVL C01482 V=800.0 PL=0
MOVL C01483 V=800.0 PL=0
MOVL C01484 V=800.0 PL=0
MOVL C01485 V=800.0 PL=0
MOVL C01486 V=800.0 PL=0
MOVL C01487 V=800.0 PL=0
MOVL C01488 V=800.0 PL=0
MOVL C01489 V=800.0 PL=0
MOVL C01490 V=800.0 PL=0
MOVL C01491 V=800.0 PL=0
MOVL C01492 V=800.0 PL=0
MOVL C01493 V=800.0 PL=0
MOVL C01494 V=800.0 PL=0
MOVL C01495 V=800.0 PL=0
MOVL C01496 V=800.0 PL=0
MOVL C01497 V=800.0 PL=0
MOVL C01498 V=800.0 PL=0
MOVL C01499 V=800.0 PL=0
MOVL C01500 V=800.0 PL=0
MOVL C01501 V=800.0 PL=0
MOVL C01502 V=800.0 PL=0
MOVL C01503 V=800.0 PL=0
MOVL C01504 V=800.0 PL=0
MOVL C01505 V=800.0 PL=0
MOVL C01506 V=800.0 PL=0
MOVL C01507 V=800.0 PL=0
MOVL C01508 V=800.0 PL=0
MOVL C01509 V=800.0 PL=0
MOVL C01510 V=800.0 PL=0
MOVL C01511 V=800.0 PL=0
MOVL C01512 V=800.0 PL=0
MOVL C01513 V=800.0 PL=0
MOVL C01514 V=800.0 PL=0
MOVL C01515 V=800.0 PL=0
MOVL C01516 V=800.0 PL=0
MOVL C01517 V=800.0 PL=0
MOVL C01518 V=800.0 PL=0
MOVL C01519 V=800.0 PL=0
MOVL C01520 V=800.0 PL=0
MOVL C01521 V=800.0 PL=0
MOVL C01522 V=800.0 PL=0
MOVL C01523 V=800.0 PL=0
MOVL C01524 V=800.0 PL=0
MOVL C01525 V=800.0 PL=0
MOVL C01526 V=800.0 PL=0
MOVL C01527 V=800.0 PL=0
MOVL C01528 V=800.0 PL=0
MOVL C01529 V=800.0 PL=0
MOVL C01530 V=800.0 PL=0
MOVL C01531 V=800.0 PL=0
MOVL C01532 V=800.0 PL=0
MOVL C01533 V=800.0 PL=0
MOVL C01534 V=800.0 PL=0
MOVL C01535 V=800.0 PL=0
MOVL C01536 V=800.0 PL=0
MOVL C01537 V=800.0 PL=0
MOVL C01538 V=800.0 PL=0
MOVL C01539 V=800.0 PL=0
MOVL C01540 V=800.0 PL=0
MOVL C01541 V=800.0 PL=0
MOVL C01542 V=800.0 PL=0
MOVL C01543 V=800.0 PL=0
MOVL C01544 V=800.0 PL=0
MOVL C01545 V=800.0 PL=0
MOVL C01546 V=800.0 PL=0
MOVL C01547 V=800.0 PL=0
MOVL C01548 V=800.0 PL=0
MOVL C01549 V=800.0 PL=0
MOVL C01550 V=800.0 PL=0
MOVL C01551 V=800.0 PL=0
MOVL C01552 V=800.0 PL=0
MOVL C01553 V=800.0 PL=0
MOVL C01554 V=800.0 PL=0
MOVL C01555 V=800.0 PL=0
MOVL C01556 V=800.0 PL=0
MOVL C01557 V=800.0 PL=0
MOVL C01558 V=800.0 PL=0
MOVL C01559 V=800.0 PL=0
MOVL C01560 V=800.0 PL=0
MOVL C01561 V=800.0 PL=0
MOVL C01562 V=800.0 PL=0
MOVL C01563 V=800.0 PL=0
MOVL C01564 V=800.0 PL=0
MOVL C01565 V=800.0 PL=0
MOVL C01566 V=800.0 PL=0
MOVL C01567 V=800.0 PL=0
MOVL C01568 V=800.0 PL=0
MOVL C01569 V=800.0 PL=0
MOVL C01570 V=800.0 PL=0
MOVL C01571 V=800.0 PL=0
MOVL C01572 V=800.0 PL=0
MOVL C01573 V=800.0 PL=0
MOVL C01574 V=800.0 PL=0
MOVL C01575 V=800.0 PL=0
MOVL C01576 V=800.0 PL=0
MOVL C01577 V=800.0 PL=0
MOVL C01578 V=800.0 PL=0
MOVL C01579 V=800.0 PL=0
MOVL C01580 V=800.0 PL=0
MOVL C01581 V=800.0 PL=0
MOVL C01582 V=800.0 PL=0
MOVL C01583 V=800.0 PL=0
MOVL C01584 V=800.0 PL=0
MOVL C01585 V=800.0 PL=0
MOVL C01586 V=800.0 PL=0
MOVL C01587 V=800.0 PL=0
MOVL C01588 V=800.0 PL=0
MOVL C01589 V=800.0 PL=0
MOVL C01590 V=800.0 PL=0
MOVL C01591 V=800.0 PL=0
MOVL C01592 V=800.0 PL=0
MOVL C01593 V=800.0 PL=0
MOVL C01594 V=800.0 PL=0
MOVL C01595 V=800.0 PL=0
MOVL C01596 V=800.0 PL=0
MOVL C01597 V=800.0 PL=0
MOVL C01598 V=800.0 PL=0
MOVL C01599 V=800.0 PL=0
MOVL C01600 V=800.0 PL=0
MOVL C01601 V=800.0 PL=0
MOVL C01602 V=800.0 PL=0
MOVL C01603 V=800.0 PL=0
MOVL C01604 V=800.0 PL=0
MOVL C01605 V=800.0 PL=0
MOVL C01606 V=800.0 PL=0
MOVL C01607 V=800.0 PL=0
MOVL C01608 V=800.0 PL=0
MOVL C01609 V=800.0 PL=0
MOVL C01610 V=800.0 PL=0
MOVL C01611 V=800.0 PL=0
MOVL C01612 V=800.0 PL=0
MOVL C01613 V=800.0 PL=0
MOVL C01614 V=800.0 PL=0
MOVL C01615 V=800.0 PL=0
MOVL C01616 V=800.0 PL=0
MOVL C01617 V=800.0 PL=0
MOVL C01618 V=800.0 PL=0
MOVL C01619 V=800.0 PL=0
MOVL C01620 V=800.0 PL=0
MOVL C01621 V=800.0 PL=0
MOVL C01622 V=800.0 PL=0
MOVL C01623 V=800.0 PL=0
MOVL C01624 V=800.0 PL=0
MOVL C01625 V=800.0 PL=0
MOVL C01626 V=800.0 PL=0
MOVL C01627 V=800.0 PL=0
MOVL C01628 V=800.0 PL=0
MOVL C01629 V=800.0 PL=0
MOVL C01630 V=800.0 PL=0
MOVL C01631 V=800.0 PL=0
MOVL C01632 V=800.0 PL=0
MOVL C01633 V=800.0 PL=0
MOVL C01634 V=800.0 PL=0
MOVL C01635 V=800.0 PL=0
MOVL C01636 V=800.0 PL=0
MOVL C01637 V=800.0 PL=0
MOVL C01638 V=800.0 PL=0
MOVL C01639 V=800.0 PL=0
MOVL C01640 V=800.0 PL=0
MOVL C01641 V=800.0 PL=0
MOVL C01642 V=800.0 PL=0
MOVL C01643 V=800.0 PL=0
MOVL C01644 V=800.0 PL=0
MOVL C01645 V=800.0 PL=0
MOVL C01646 V=800.0 PL=0
MOVL C01647 V=800.0 PL=0
MOVL C01648 V=800.0 PL=0
MOVL C01649 V=800.0 PL=0
MOVL C01650 V=800.0 PL=0
MOVL C01651 V=800.0 PL=0
MOVL C01652 V=800.0 PL=0
MOVL C01653 V=800.0 PL=0
MOVL C01654 V=800.0 PL=0
MOVL C01655 V=800.0 PL=0
MOVL C01656 V=800.0 PL=0
MOVL C01657 V=800.0 PL=0
MOVL C01658 V=800.0 PL=0
MOVL C01659 V=800.0 PL=0
MOVL C01660 V=800.0 PL=0
MOVL C01661 V=800.0 PL=0
MOVL C01662 V=800.0 PL=0
MOVL C01663 V=800.0 PL=0
MOVL C01664 V=800.0 PL=0
MOVL C01665 V=800.0 PL=0
MOVL C01666 V=800.0 PL=0
MOVL C01667 V=800.0 PL=0
MOVL C01668 V=800.0 PL=0
MOVL C01669 V=800.0 PL=0
MOVL C01670 V=800.0 PL=0
MOVL C01671 V=800.0 PL=0
MOVL C01672 V=800.0 PL=0
MOVL C01673 V=800.0 PL=0
MOVL C01674 V=800.0 PL=0
MOVL C01675 V=800.0 PL=0
MOVL C01676 V=800.0 PL=0
MOVL C01677 V=800.0 PL=0
MOVL C01678 V=800.0 PL=0
MOVL C01679 V=800.0 PL=0
MOVL C01680 V=800.0 PL=0
MOVL C01681 V=800.0 PL=0
MOVL C01682 V=800.0 PL=0
MOVL C01683 V=800.0 PL=0
MOVL C01684 V=800.0 PL=0
MOVL C01685 V=800.0 PL=0
MOVL C01686 V=800.0 PL=0
MOVL C01687 V=800.0 PL=0
MOVL C01688 V=800.0 PL=0
MOVL C01689 V=800.0 PL=0
MOVL C01690 V=800.0 PL=0
MOVL C01691 V=800.0 PL=0
MOVL C01692 V=800.0 PL=0
MOVL C01693 V=800.0 PL=0
MOVL C01694 V=800.0 PL=0
MOVL C01695 V=800.0 PL=0
MOVL C01696 V=800.0 PL=0
MOVL C01697 V=800.0 PL=0
MOVL C01698 V=800.0 PL=0
MOVL C01699 V=800.0 PL=0
MOVL C01700 V=800.0 PL=0
MOVL C01701 V=800.0 PL=0
MOVL C01702 V=800.0 PL=0
MOVL C01703 V=800.0 PL=0
MOVL C01704 V=800.0 PL=0
MOVL C01705 V=800.0 PL=0
MOVL C01706 V=800.0 PL=0
MOVL C01707 V=800.0 PL=0
MOVL C01708 V=800.0 PL=0
MOVL C01709 V=800.0 PL=0
MOVL C01710 V=800.0 PL=0
MOVL C01711 V=800.0 PL=0
MOVL C01712 V=800.0 PL=0
MOVL C01713 V=800.0 PL=0
MOVL C01714 V=800.0 PL=0
MOVL C01715 V=800.0 PL=0
MOVL C01716 V=800.0 PL=0
MOVL C01717 V=800.0 PL=0
MOVL C01718 V=800.0 PL=0
MOVL C01719 V=800.0 PL=0
MOVL C01720 V=800.0 PL=0
MOVL C01721 V=800.0 PL=0
MOVL C01722 V=800.0 PL=0
MOVL C01723 V=800.0 PL=0
MOVL C01724 V=800.0 PL=0
MOVL C01725 V=800.0 PL=0
MOVL C01726 V=800.0 PL=0
MOVL C01727 V=800.0 PL=0
MOVL C01728 V=800.0 PL=0
MOVL C01729 V=800.0 PL=0
MOVL C01730 V=800.0 PL=0
MOVL C01731 V=800.0 PL=0
MOVL C01732 V=800.0 PL=0
MOVL C01733 V=800.0 PL=0
MOVL C01734 V=800.0 PL=0
MOVL C01735 V=800.0 PL=0
MOVL C01736 V=800.0 PL=0
MOVL C01737 V=800.0 PL=0
MOVL C01738 V=800.0 PL=0
MOVL C01739 V=800.0 PL=0
MOVL C01740 V=800.0 PL=0
MOVL C01741 V=800.0 PL=0
MOVL C01742 V=800.0 PL=0
MOVL C01743 V=800.0 PL=0
MOVL C01744 V=800.0 PL=0
MOVL C01745 V=800.0 PL=0
MOVL C01746 V=800.0 PL=0
MOVL C01747 V=800.0 PL=0
MOVL C01748 V=800.0 PL=0
MOVL C01749 V=800.0 PL=0
MOVL C01750 V=800.0 PL=0
MOVL C01751 V=800.0 PL=0
MOVL C01752 V=800.0 PL=0
MOVL C01753 V=800.0 PL=0
MOVL C01754 V=800.0 PL=0
MOVL C01755 V=800.0 PL=0
MOVL C01756 V=800.0 PL=0
MOVL C01757 V=800.0 PL=0
MOVL C01758 V=800.0 PL=0
MOVL C01759 V=800.0 PL=0
MOVL C01760 V=800.0 PL=0
MOVL C01761 V=800.0 PL=0
MOVL C01762 V=800.0 PL=0
MOVL C01763 V=800.0 PL=0
MOVL C01764 V=800.0 PL=0
MOVL C01765 V=800.0 PL=0
MOVL C01766 V=800.0 PL=0
MOVL C01767 V=800.0 PL=0
MOVL C01768 V=800.0 PL=0
MOVL C01769 V=800.0 PL=0
MOVL C01770 V=800.0 PL=0
MOVL C01771 V=800.0 PL=0
MOVL C01772 V=800.0 PL=0
MOVL C01773 V=800.0 PL=0
MOVL C01774 V=800.0 PL=0
MOVL C01775 V=800.0 PL=0
MOVL C01776 V=800.0 PL=0
MOVL C01777 V=800.0 PL=0
MOVL C01778 V=800.0 PL=0
MOVL C01779 V=800.0 PL=0
MOVL C01780 V=800.0 PL=0
MOVL C01781 V=800.0 PL=0
MOVL C01782 V=800.0 PL=0
MOVL C01783 V=800.0 PL=0
MOVL C01784 V=800.0 PL=0
MOVL C01785 V=800.0 PL=0
MOVL C01786 V=800.0 PL=0
MOVL C01787 V=800.0 PL=0
MOVL C01788 V=800.0 PL=0
MOVL C01789 V=800.0 PL=0
MOVL C01790 V=800.0 PL=0
MOVL C01791 V=800.0 PL=0
MOVL C01792 V=800.0 PL=0
MOVL C01793 V=800.0 PL=0
MOVL C01794 V=800.0 PL=0
MOVL C01795 V=800.0 PL=0
MOVL C01796 V=800.0 PL=0
MOVL C01797 V=800.0 PL=0
MOVL C01798 V=800.0 PL=0
MOVL C01799 V=800.0 PL=0
MOVL C01800 V=800.0 PL=0
MOVL C01801 V=800.0 PL=0
MOVL C01802 V=800.0 PL=0
MOVL C01803 V=800.0 PL=0
MOVL C01804 V=800.0 PL=0
MOVL C01805 V=800.0 PL=0
MOVL C01806 V=800.0 PL=0
MOVL C01807 V=800.0 PL=0
MOVL C01808 V=800.0 PL=0
MOVL C01809 V=800.0 PL=0
MOVL C01810 V=800.0 PL=0
MOVL C01811 V=800.0 PL=0
MOVL C01812 V=800.0 PL=0
MOVL C01813 V=800.0 PL=0
MOVL C01814 V=800.0 PL=0
MOVL C01815 V=800.0 PL=0
MOVL C01816 V=800.0 PL=0
MOVL C01817 V=800.0 PL=0
MOVL C01818 V=800.0 PL=0
MOVL C01819 V=800.0 PL=0
MOVL C01820 V=800.0 PL=0
MOVL C01821 V=800.0 PL=0
MOVL C01822 V=800.0 PL=0
MOVL C01823 V=800.0 PL=0
MOVL C01824 V=800.0 PL=0
MOVL C01825 V=800.0 PL=0
MOVL C01826 V=800.0 PL=0
MOVL C01827 V=800.0 PL=0
MOVL C01828 V=800.0 PL=0
MOVL C01829 V=800.0 PL=0
MOVL C01830 V=800.0 PL=0
MOVL C01831 V=800.0 PL=0
MOVL C01832 V=800.0 PL=0
MOVL C01833 V=800.0 PL=0
MOVL C01834 V=800.0 PL=0
MOVL C01835 V=800.0 PL=0
MOVL C01836 V=800.0 PL=0
MOVL C01837 V=800.0 PL=0
MOVL C01838 V=800.0 PL=0
MOVL C01839 V=800.0 PL=0
MOVL C01840 V=800.0 PL=0
MOVL C01841 V=800.0 PL=0
MOVL C01842 V=800.0 PL=0
MOVL C01843 V=800.0 PL=0
MOVL C01844 V=800.0 PL=0
MOVL C01845 V=800.0 PL=0
MOVL C01846 V=800.0 PL=0
MOVL C01847 V=800.0 PL=0
MOVL C01848 V=800.0 PL=0
MOVL C01849 V=800.0 PL=0
MOVL C01850 V=800.0 PL=0
MOVL C01851 V=800.0 PL=0
MOVL C01852 V=800.0 PL=0
MOVL C01853 V=800.0 PL=0
MOVL C01854 V=800.0 PL=0
MOVL C01855 V=800.0 PL=0
MOVL C01856 V=800.0 PL=0
MOVL C01857 V=800.0 PL=0
MOVL C01858 V=800.0 PL=0
MOVL C01859 V=800.0 PL=0
MOVL C01860 V=800.0 PL=0
MOVL C01861 V=800.0 PL=0
MOVL C01862 V=800.0 PL=0
MOVL C01863 V=800.0 PL=0
MOVL C01864 V=800.0 PL=0
MOVL C01865 V=800.0 PL=0
MOVL C01866 V=800.0 PL=0
MOVL C01867 V=800.0 PL=0
MOVL C01868 V=800.0 PL=0
MOVL C01869 V=800.0 PL=0
MOVL C01870 V=800.0 PL=0
MOVL C01871 V=800.0 PL=0
MOVL C01872 V=800.0 PL=0
MOVL C01873 V=800.0 PL=0
MOVL C01874 V=800.0 PL=0
MOVL C01875 V=800.0 PL=0
MOVL C01876 V=800.0 PL=0
MOVL C01877 V=800.0 PL=0
MOVL C01878 V=800.0 PL=0
MOVL C01879 V=800.0 PL=0
MOVL C01880 V=800.0 PL=0
MOVL C01881 V=800.0 PL=0
MOVL C01882 V=800.0 PL=0
MOVL C01883 V=800.0 PL=0
MOVL C01884 V=800.0 PL=0
MOVL C01885 V=800.0 PL=0
MOVL C01886 V=800.0 PL=0
MOVL C01887 V=800.0 PL=0
MOVL C01888 V=800.0 PL=0
MOVL C01889 V=800.0 PL=0
MOVL C01890 V=800.0 PL=0
MOVL C01891 V=800.0 PL=0
MOVL C01892 V=800.0 PL=0
MOVL C01893 V=800.0 PL=0
MOVL C01894 V=800.0 PL=0
MOVL C01895 V=800.0 PL=0
MOVL C01896 V=800.0 PL=0
MOVL C01897 V=800.0 PL=0
MOVL C01898 V=800.0 PL=0
MOVL C01899 V=800.0 PL=0
MOVL C01900 V=800.0 PL=0
MOVL C01901 V=800.0 PL=0
MOVL C01902 V=800.0 PL=0
MOVL C01903 V=800.0 PL=0
MOVL C01904 V=800.0 PL=0
MOVL C01905 V=800.0 PL=0
MOVL C01906 V=800.0 PL=0
MOVL C01907 V=800.0 PL=0
MOVL C01908 V=800.0 PL=0
MOVL C01909 V=800.0 PL=0
MOVL C01910 V=800.0 PL=0
MOVL C01911 V=800.0 PL=0
MOVL C01912 V=800.0 PL=0
MOVL C01913 V=800.0 PL=0
MOVL C01914 V=800.0 PL=0
MOVL C01915 V=800.0 PL=0
MOVL C01916 V=800.0 PL=0
MOVL C01917 V=800.0 PL=0
MOVL C01918 V=800.0 PL=0
MOVL C01919 V=800.0 PL=0
MOVL C01920 V=800.0 PL=0
MOVL C01921 V=800.0 PL=0
MOVL C01922 V=800.0 PL=0
MOVL C01923 V=800.0 PL=0
MOVL C01924 V=800.0 PL=0
MOVL C01925 V=800.0 PL=0
MOVL C01926 V=800.0 PL=0
MOVL C01927 V=800.0 PL=0
MOVL C01928 V=800.0 PL=0
MOVL C01929 V=800.0 PL=0
MOVL C01930 V=800.0 PL=0
MOVL C01931 V=800.0 PL=0
MOVL C01932 V=800.0 PL=0
MOVL C01933 V=800.0 PL=0
MOVL C01934 V=800.0 PL=0
MOVL C01935 V=800.0 PL=0
MOVL C01936 V=800.0 PL=0
MOVL C01937 V=800.0 PL=0
MOVL C01938 V=800.0 PL=0
MOVL C01939 V=800.0 PL=0
MOVL C01940 V=800.0 PL=0
MOVL C01941 V=800.0 PL=0
MOVL C01942 V=800.0 PL=0
MOVL C01943 V=800.0 PL=0
MOVL C01944 V=800.0 PL=0
MOVL C01945 V=800.0 PL=0
MOVL C01946 V=800.0 PL=0
MOVL C01947 V=800.0 PL=0
MOVL C01948 V=800.0 PL=0
MOVL C01949 V=800.0 PL=0
MOVL C01950 V=800.0 PL=0
MOVL C01951 V=800.0 PL=0
MOVL C01952 V=800.0 PL=0
MOVL C01953 V=800.0 PL=0
MOVL C01954 V=800.0 PL=0
MOVL C01955 V=800.0 PL=0
MOVL C01956 V=800.0 PL=0
MOVL C01957 V=800.0 PL=0
MOVL C01958 V=800.0 PL=0
MOVL C01959 V=800.0 PL=0
MOVL C01960 V=800.0 PL=0
MOVL C01961 V=800.0 PL=0
MOVL C01962 V=800.0 PL=0
MOVL C01963 V=800.0 PL=0
MOVL C01964 V=800.0 PL=0
MOVL C01965 V=800.0 PL=0
MOVL C01966 V=800.0 PL=0
MOVL C01967 V=800.0 PL=0
MOVL C01968 V=800.0 PL=0
MOVL C01969 V=800.0 PL=0
MOVL C01970 V=800.0 PL=0
MOVL C01971 V=800.0 PL=0
MOVL C01972 V=800.0 PL=0
MOVL C01973 V=800.0 PL=0
MOVL C01974 V=800.0 PL=0
MOVL C01975 V=800.0 PL=0
MOVL C01976 V=800.0 PL=0
MOVL C01977 V=800.0 PL=0
MOVL C01978 V=800.0 PL=0
MOVL C01979 V=800.0 PL=0
MOVL C01980 V=800.0 PL=0
MOVL C01981 V=800.0 PL=0
MOVL C01982 V=800.0 PL=0
MOVL C01983 V=800.0 PL=0
MOVL C01984 V=800.0 PL=0
MOVL C01985 V=800.0 PL=0
MOVL C01986 V=800.0 PL=0
MOVL C01987 V=800.0 PL=0
MOVL C01988 V=800.0 PL=0
MOVL C01989 V=800.0 PL=0
MOVL C01990 V=800.0 PL=0
MOVL C01991 V=800.0 PL=0
MOVL C01992 V=800.0 PL=0
MOVL C01993 V=800.0 PL=0
MOVL C01994 V=800.0 PL=0
MOVL C01995 V=800.0 PL=0
MOVL C01996 V=800.0 PL=0
MOVL C01997 V=800.0 PL=0
MOVL C01998 V=800.0 PL=0
MOVL C01999 V=800.0 PL=0
MOVL C02000 V=800.0 PL=0
MOVL C02001 V=800.0 PL=0
MOVL C02002 V=800.0 PL=0
MOVL C02003 V=800.0 PL=0
MOVL C02004 V=800.0 PL=0
MOVL C02005 V=800.0 PL=0
MOVL C02006 V=800.0 PL=0
MOVL C02007 V=800.0 PL=0
MOVL C02008 V=800.0 PL=0
MOVL C02009 V=800.0 PL=0
MOVL C02010 V=800.0 PL=0
MOVL C02011 V=800.0 PL=0
MOVL C02012 V=800.0 PL=0
MOVL C02013 V=800.0 PL=0
MOVL C02014 V=800.0 PL=0
MOVL C02015 V=800.0 PL=0
MOVL C02016 V=800.0 PL=0
MOVL C02017 V=800.0 PL=0
MOVL C02018 V=800.0 PL=0
MOVL C02019 V=800.0 PL=0
MOVL C02020 V=800.0 PL=0
MOVL C02021 V=800.0 PL=0
MOVL C02022 V=800.0 PL=0
MOVL C02023 V=800.0 PL=0
MOVL C02024 V=800.0 PL=0
MOVL C02025 V=800.0 PL=0
MOVL C02026 V=800.0 PL=0
MOVL C02027 V=800.0 PL=0
MOVL C02028 V=800.0 PL=0
MOVL C02029 V=800.0 PL=0
MOVL C02030 V=800.0 PL=0
MOVL C02031 V=800.0 PL=0
MOVL C02032 V=800.0 PL=0
MOVL C02033 V=800.0 PL=0
MOVL C02034 V=800.0 PL=0
MOVL C02035 V=800.0 PL=0
MOVL C02036 V=800.0 PL=0
MOVL C02037 V=800.0 PL=0
MOVL C02038 V=800.0 PL=0
MOVL C02039 V=800.0 PL=0
MOVL C02040 V=800.0 PL=0
MOVL C02041 V=800.0 PL=0
MOVL C02042 V=800.0 PL=0
MOVL C02043 V=800.0 PL=0
MOVL C02044 V=800.0 PL=0
MOVL C02045 V=800.0 PL=0
MOVL C02046 V=800.0 PL=0
MOVL C02047 V=800.0 PL=0
MOVL C02048 V=800.0 PL=0
MOVL C02049 V=800.0 PL=0
MOVL C02050 V=800.0 PL=0
MOVL C02051 V=800.0 PL=0
MOVL C02052 V=800.0 PL=0
MOVL C02053 V=800.0 PL=0
MOVL C02054 V=800.0 PL=0
MOVL C02055 V=800.0 PL=0
MOVL C02056 V=800.0 PL=0
MOVL C02057 V=800.0 PL=0
MOVL C02058 V=800.0 PL=0
MOVL C02059 V=800.0 PL=0
MOVL C02060 V=800.0 PL=0
MOVL C02061 V=800.0 PL=0
MOVL C02062 V=800.0 PL=0
MOVL C02063 V=800.0 PL=0
MOVL C02064 V=800.0 PL=0
MOVL C02065 V=800.0 PL=0
MOVL C02066 V=800.0 PL=0
MOVL C02067 V=800.0 PL=0
MOVL C02068 V=800.0 PL=0
MOVL C02069 V=800.0 PL=0
MOVL C02070 V=800.0 PL=0
MOVL C02071 V=800.0 PL=0
MOVL C02072 V=800.0 PL=0
MOVL C02073 V=800.0 PL=0
MOVL C02074 V=800.0 PL=0
MOVL C02075 V=800.0 PL=0
MOVL C02076 V=800.0 PL=0
MOVL C02077 V=800.0 PL=0
MOVL C02078 V=800.0 PL=0
MOVL C02079 V=800.0 PL=0
MOVL C02080 V=800.0 PL=0
MOVL C02081 V=800.0 PL=0
MOVL C02082 V=800.0 PL=0
MOVL C02083 V=800.0 PL=0
MOVL C02084 V=800.0 PL=0
MOVL C02085 V=800.0 PL=0
MOVL C02086 V=800.0 PL=0
MOVL C02087 V=800.0 PL=0
MOVL C02088 V=800.0 PL=0
MOVL C02089 V=800.0 PL=0
MOVL C02090 V=800.0 PL=0
MOVL C02091 V=800.0 PL=0
MOVL C02092 V=800.0 PL=0
MOVL C02093 V=800.0 PL=0
MOVL C02094 V=800.0 PL=0
MOVL C02095 V=800.0 PL=0
MOVL C02096 V=800.0 PL=0
MOVL C02097 V=800.0 PL=0
MOVL C02098 V=800.0 PL=0
MOVL C02099 V=800.0 PL=0
MOVL C02100 V=800.0 PL=0
MOVL C02101 V=800.0 PL=0
MOVL C02102 V=800.0 PL=0
MOVL C02103 V=800.0 PL=0
MOVL C02104 V=800.0 PL=0
MOVL C02105 V=800.0 PL=0
MOVL C02106 V=800.0 PL=0
MOVL C02107 V=800.0 PL=0
MOVL C02108 V=800.0 PL=0
MOVL C02109 V=800.0 PL=0
MOVL C02110 V=800.0 PL=0
MOVL C02111 V=800.0 PL=0
MOVL C02112 V=800.0 PL=0
MOVL C02113 V=800.0 PL=0
MOVL C02114 V=800.0 PL=0
MOVL C02115 V=800.0 PL=0
MOVL C02116 V=800.0 PL=0
MOVL C02117 V=800.0 PL=0
MOVL C02118 V=800.0 PL=0
MOVL C02119 V=800.0 PL=0
MOVL C02120 V=800.0 PL=0
MOVL C02121 V=800.0 PL=0
MOVL C02122 V=800.0 PL=0
MOVL C02123 V=800.0 PL=0
MOVL C02124 V=800.0 PL=0
MOVL C02125 V=800.0 PL=0
MOVL C02126 V=800.0 PL=0
MOVL C02127 V=800.0 PL=0
MOVL C02128 V=800.0 PL=0
MOVL C02129 V=800.0 PL=0
MOVL C02130 V=800.0 PL=0
MOVL C02131 V=800.0 PL=0
MOVL C02132 V=800.0 PL=0
MOVL C02133 V=800.0 PL=0
MOVL C02134 V=800.0 PL=0
MOVL C02135 V=800.0 PL=0
MOVL C02136 V=800.0 PL=0
MOVL C02137 V=800.0 PL=0
MOVL C02138 V=800.0 PL=0
MOVL C02139 V=800.0 PL=0
MOVL C02140 V=800.0 PL=0
MOVL C02141 V=800.0 PL=0
MOVL C02142 V=800.0 PL=0
MOVL C02143 V=800.0 PL=0
MOVL C02144 V=800.0 PL=0
MOVL C02145 V=800.0 PL=0
MOVL C02146 V=800.0 PL=0
MOVL C02147 V=800.0 PL=0
MOVL C02148 V=800.0 PL=0
MOVL C02149 V=800.0 PL=0
MOVL C02150 V=800.0 PL=0
MOVL C02151 V=800.0 PL=0
MOVL C02152 V=800.0 PL=0
MOVL C02153 V=800.0 PL=0
MOVL C02154 V=800.0 PL=0
MOVL C02155 V=800.0 PL=0
MOVL C02156 V=800.0 PL=0
MOVL C02157 V=800.0 PL=0
MOVL C02158 V=800.0 PL=0
MOVL C02159 V=800.0 PL=0
MOVL C02160 V=800.0 PL=0
MOVL C02161 V=800.0 PL=0
MOVL C02162 V=800.0 PL=0
MOVL C02163 V=800.0 PL=0
MOVL C02164 V=800.0 PL=0
MOVL C02165 V=800.0 PL=0
MOVL C02166 V=800.0 PL=0
MOVL C02167 V=800.0 PL=0
MOVL C02168 V=800.0 PL=0
MOVL C02169 V=800.0 PL=0
MOVL C02170 V=800.0 PL=0
MOVL C02171 V=800.0 PL=0
MOVL C02172 V=800.0 PL=0
MOVL C02173 V=800.0 PL=0
MOVL C02174 V=800.0 PL=0
MOVL C02175 V=800.0 PL=0
MOVL C02176 V=800.0 PL=0
MOVL C02177 V=800.0 PL=0
MOVL C02178 V=800.0 PL=0
MOVL C02179 V=800.0 PL=0
MOVL C02180 V=800.0 PL=0
MOVL C02181 V=800.0 PL=0
MOVL C02182 V=800.0 PL=0
MOVL C02183 V=800.0 PL=0
MOVL C02184 V=800.0 PL=0
MOVL C02185 V=800.0 PL=0
MOVL C02186 V=800.0 PL=0
MOVL C02187 V=800.0 PL=0
MOVL C02188 V=800.0 PL=0
MOVL C02189 V=800.0 PL=0
MOVL C02190 V=800.0 PL=0
MOVL C02191 V=800.0 PL=0
MOVL C02192 V=800.0 PL=0
MOVL C02193 V=800.0 PL=0
MOVL C02194 V=800.0 PL=0
MOVL C02195 V=800.0 PL=0
MOVL C02196 V=800.0 PL=0
MOVL C02197 V=800.0 PL=0
MOVL C02198 V=800.0 PL=0
MOVL C02199 V=800.0 PL=0
MOVL C02200 V=800.0 PL=0
MOVL C02201 V=800.0 PL=0
MOVL C02202 V=800.0 PL=0
MOVL C02203 V=800.0 PL=0
MOVL C02204 V=800.0 PL=0
MOVL C02205 V=800.0 PL=0
MOVL C02206 V=800.0 PL=0
MOVL C02207 V=800.0 PL=0
MOVL C02208 V=800.0 PL=0
MOVL C02209 V=800.0 PL=0
MOVL C02210 V=800.0 PL=0
MOVL C02211 V=800.0 PL=0
MOVL C02212 V=800.0 PL=0
MOVL C02213 V=800.0 PL=0
MOVL C02214 V=800.0 PL=0
MOVL C02215 V=800.0 PL=0
MOVL C02216 V=800.0 PL=0
MOVL C02217 V=800.0 PL=0
MOVL C02218 V=800.0 PL=0
MOVL C02219 V=800.0 PL=0
MOVL C02220 V=800.0 PL=0
MOVL C02221 V=800.0 PL=0
MOVL C02222 V=800.0 PL=0
MOVL C02223 V=800.0 PL=0
MOVL C02224 V=800.0 PL=0
MOVL C02225 V=800.0 PL=0
MOVL C02226 V=800.0 PL=0
MOVL C02227 V=800.0 PL=0
MOVL C02228 V=800.0 PL=0
MOVL C02229 V=800.0 PL=0
MOVL C02230 V=800.0 PL=0
MOVL C02231 V=800.0 PL=0
MOVL C02232 V=800.0 PL=0
MOVL C02233 V=800.0 PL=0
MOVL C02234 V=800.0 PL=0
MOVL C02235 V=800.0 PL=0
MOVL C02236 V=800.0 PL=0
MOVL C02237 V=800.0 PL=0
MOVL C02238 V=800.0 PL=0
MOVL C02239 V=800.0 PL=0
MOVL C02240 V=800.0 PL=0
MOVL C02241 V=800.0 PL=0
MOVL C02242 V=800.0 PL=0
MOVL C02243 V=800.0 PL=0
MOVL C02244 V=800.0 PL=0
MOVL C02245 V=800.0 PL=0
MOVL C02246 V=800.0 PL=0
MOVL C02247 V=800.0 PL=0
MOVL C02248 V=800.0 PL=0
MOVL C02249 V=800.0 PL=0
MOVL C02250 V=800.0 PL=0
MOVL C02251 V=800.0 PL=0
MOVL C02252 V=800.0 PL=0
MOVL C02253 V=800.0 PL=0
MOVL C02254 V=800.0 PL=0
MOVL C02255 V=800.0 PL=0
MOVL C02256 V=800.0 PL=0
MOVL C02257 V=800.0 PL=0
MOVL C02258 V=800.0 PL=0
MOVL C02259 V=800.0 PL=0
MOVL C02260 V=800.0 PL=0
MOVL C02261 V=800.0 PL=0
MOVL C02262 V=800.0 PL=0
MOVL C02263 V=800.0 PL=0
MOVL C02264 V=800.0 PL=0
MOVL C02265 V=800.0 PL=0
MOVL C02266 V=800.0 PL=0
MOVL C02267 V=800.0 PL=0
MOVL C02268 V=800.0 PL=0
MOVL C02269 V=800.0 PL=0
MOVL C02270 V=800.0 PL=0
MOVL C02271 V=800.0 PL=0
MOVL C02272 V=800.0 PL=0
MOVL C02273 V=800.0 PL=0
MOVL C02274 V=800.0 PL=0
MOVL C02275 V=800.0 PL=0
MOVL C02276 V=800.0 PL=0
MOVL C02277 V=800.0 PL=0
MOVL C02278 V=800.0 PL=0
MOVL C02279 V=800.0 PL=0
MOVL C02280 V=800.0 PL=0
MOVL C02281 V=800.0 PL=0
MOVL C02282 V=800.0 PL=0
MOVL C02283 V=800.0 PL=0
MOVL C02284 V=800.0 PL=0
MOVL C02285 V=800.0 PL=0
MOVL C02286 V=800.0 PL=0
MOVL C02287 V=800.0 PL=0
MOVL C02288 V=800.0 PL=0
MOVL C02289 V=800.0 PL=0
MOVL C02290 V=800.0 PL=0
MOVL C02291 V=800.0 PL=0
MOVL C02292 V=800.0 PL=0
MOVL C02293 V=800.0 PL=0
MOVL C02294 V=800.0 PL=0
MOVL C02295 V=800.0 PL=0
MOVL C02296 V=800.0 PL=0
MOVL C02297 V=800.0 PL=0
MOVL C02298 V=800.0 PL=0
MOVL C02299 V=800.0 PL=0
MOVL C02300 V=800.0 PL=0
MOVL C02301 V=800.0 PL=0
MOVL C02302 V=800.0 PL=0
MOVL C02303 V=800.0 PL=0
MOVL C02304 V=800.0 PL=0
MOVL C02305 V=800.0 PL=0
MOVL C02306 V=800.0 PL=0
MOVL C02307 V=800.0 PL=0
MOVL C02308 V=800.0 PL=0
MOVL C02309 V=800.0 PL=0
MOVL C02310 V=800.0 PL=0
MOVL C02311 V=800.0 PL=0
MOVL C02312 V=800.0 PL=0
MOVL C02313 V=800.0 PL=0
MOVL C02314 V=800.0 PL=0
MOVL C02315 V=800.0 PL=0
MOVL C02316 V=800.0 PL=0
MOVL C02317 V=800.0 PL=0
MOVL C02318 V=800.0 PL=0
MOVL C02319 V=800.0 PL=0
MOVL C02320 V=800.0 PL=0
MOVL C02321 V=800.0 PL=0
MOVL C02322 V=800.0 PL=0
MOVL C02323 V=800.0 PL=0
MOVL C02324 V=800.0 PL=0
MOVL C02325 V=800.0 PL=0
MOVL C02326 V=800.0 PL=0
MOVL C02327 V=800.0 PL=0
MOVL C02328 V=800.0 PL=0
MOVL C02329 V=800.0 PL=0
MOVL C02330 V=800.0 PL=0
MOVL C02331 V=800.0 PL=0
MOVL C02332 V=800.0 PL=0
MOVL C02333 V=800.0 PL=0
MOVL C02334 V=800.0 PL=0
MOVL C02335 V=800.0 PL=0
MOVL C02336 V=800.0 PL=0
MOVL C02337 V=800.0 PL=0
MOVL C02338 V=800.0 PL=0
MOVL C02339 V=800.0 PL=0
MOVL C02340 V=800.0 PL=0
MOVL C02341 V=800.0 PL=0
MOVL C02342 V=800.0 PL=0
MOVL C02343 V=800.0 PL=0
MOVL C02344 V=800.0 PL=0
MOVL C02345 V=800.0 PL=0
MOVL C02346 V=800.0 PL=0
MOVL C02347 V=800.0 PL=0
MOVL C02348 V=800.0 PL=0
MOVL C02349 V=800.0 PL=0
MOVL C02350 V=800.0 PL=0
MOVL C02351 V=800.0 PL=0
MOVL C02352 V=800.0 PL=0
MOVL C02353 V=800.0 PL=0
MOVL C02354 V=800.0 PL=0
MOVL C02355 V=800.0 PL=0
MOVL C02356 V=800.0 PL=0
MOVL C02357 V=800.0 PL=0
MOVL C02358 V=800.0 PL=0
MOVL C02359 V=800.0 PL=0
MOVL C02360 V=800.0 PL=0
MOVL C02361 V=800.0 PL=0
MOVL C02362 V=800.0 PL=0
MOVL C02363 V=800.0 PL=0
MOVL C02364 V=800.0 PL=0
MOVL C02365 V=800.0 PL=0
MOVL C02366 V=800.0 PL=0
MOVL C02367 V=800.0 PL=0
MOVL C02368 V=800.0 PL=0
MOVL C02369 V=800.0 PL=0
MOVL C02370 V=800.0 PL=0
MOVL C02371 V=800.0 PL=0
MOVL C02372 V=800.0 PL=0
MOVL C02373 V=800.0 PL=0
MOVL C02374 V=800.0 PL=0
MOVL C02375 V=800.0 PL=0
MOVL C02376 V=800.0 PL=0
MOVL C02377 V=800.0 PL=0
MOVL C02378 V=800.0 PL=0
MOVL C02379 V=800.0 PL=0
MOVL C02380 V=800.0 PL=0
MOVL C02381 V=800.0 PL=0
MOVL C02382 V=800.0 PL=0
MOVL C02383 V=800.0 PL=0
MOVL C02384 V=800.0 PL=0
MOVL C02385 V=800.0 PL=0
MOVL C02386 V=800.0 PL=0
MOVL C02387 V=800.0 PL=0
MOVL C02388 V=800.0 PL=0
MOVL C02389 V=800.0 PL=0
MOVL C02390 V=800.0 PL=0
MOVL C02391 V=800.0 PL=0
MOVL C02392 V=800.0 PL=0
MOVL C02393 V=800.0 PL=0
MOVL C02394 V=800.0 PL=0
MOVL C02395 V=800.0 PL=0
MOVL C02396 V=800.0 PL=0
MOVL C02397 V=800.0 PL=0
MOVL C02398 V=800.0 PL=0
MOVL C02399 V=800.0 PL=0
MOVL C02400 V=800.0 PL=0
MOVL C02401 V=800.0 PL=0
MOVL C02402 V=800.0 PL=0
MOVL C02403 V=800.0 PL=0
MOVL C02404 V=800.0 PL=0
MOVL C02405 V=800.0 PL=0
MOVL C02406 V=800.0 PL=0
MOVL C02407 V=800.0 PL=0
MOVL C02408 V=800.0 PL=0
MOVL C02409 V=800.0 PL=0
MOVL C02410 V=800.0 PL=0
MOVL C02411 V=800.0 PL=0
MOVL C02412 V=800.0 PL=0
MOVL C02413 V=800.0 PL=0
MOVL C02414 V=800.0 PL=0
MOVL C02415 V=800.0 PL=0
MOVL C02416 V=800.0 PL=0
MOVL C02417 V=800.0 PL=0
MOVL C02418 V=800.0 PL=0
MOVL C02419 V=800.0 PL=0
MOVL C02420 V=800.0 PL=0
MOVL C02421 V=800.0 PL=0
MOVL C02422 V=800.0 PL=0
MOVL C02423 V=800.0 PL=0
MOVL C02424 V=800.0 PL=0
MOVL C02425 V=800.0 PL=0
MOVL C02426 V=800.0 PL=0
MOVL C02427 V=800.0 PL=0
MOVL C02428 V=800.0 PL=0
MOVL C02429 V=800.0 PL=0
MOVL C02430 V=800.0 PL=0
MOVL C02431 V=800.0 PL=0
MOVL C02432 V=800.0 PL=0
MOVL C02433 V=800.0 PL=0
MOVL C02434 V=800.0 PL=0
MOVL C02435 V=800.0 PL=0
MOVL C02436 V=800.0 PL=0
MOVL C02437 V=800.0 PL=0
MOVL C02438 V=800.0 PL=0
MOVL C02439 V=800.0 PL=0
MOVL C02440 V=800.0 PL=0
MOVL C02441 V=800.0 PL=0
MOVL C02442 V=800.0 PL=0
MOVL C02443 V=800.0 PL=0
MOVL C02444 V=800.0 PL=0
MOVL C02445 V=800.0 PL=0
MOVL C02446 V=800.0 PL=0
MOVL C02447 V=800.0 PL=0
MOVL C02448 V=800.0 PL=0
MOVL C02449 V=800.0 PL=0
MOVL C02450 V=800.0 PL=0
MOVL C02451 V=800.0 PL=0
MOVL C02452 V=800.0 PL=0
MOVL C02453 V=800.0 PL=0
MOVL C02454 V=800.0 PL=0
MOVL C02455 V=800.0 PL=0
MOVL C02456 V=800.0 PL=0
MOVL C02457 V=800.0 PL=0
MOVL C02458 V=800.0 PL=0
MOVL C02459 V=800.0 PL=0
MOVL C02460 V=800.0 PL=0
MOVL C02461 V=800.0 PL=0
MOVL C02462 V=800.0 PL=0
MOVL C02463 V=800.0 PL=0
MOVL C02464 V=800.0 PL=0
MOVL C02465 V=800.0 PL=0
MOVL C02466 V=800.0 PL=0
MOVL C02467 V=800.0 PL=0
MOVL C02468 V=800.0 PL=0
MOVL C02469 V=800.0 PL=0
MOVL C02470 V=800.0 PL=0
MOVL C02471 V=800.0 PL=0
MOVL C02472 V=800.0 PL=0
MOVL C02473 V=800.0 PL=0
MOVL C02474 V=800.0 PL=0
MOVL C02475 V=800.0 PL=0
MOVL C02476 V=800.0 PL=0
MOVL C02477 V=800.0 PL=0
MOVL C02478 V=800.0 PL=0
MOVL C02479 V=800.0 PL=0
MOVL C02480 V=800.0 PL=0
MOVL C02481 V=800.0 PL=0
MOVL C02482 V=800.0 PL=0
MOVL C02483 V=800.0 PL=0
MOVL C02484 V=800.0 PL=0
MOVL C02485 V=800.0 PL=0
MOVL C02486 V=800.0 PL=0
MOVL C02487 V=800.0 PL=0
MOVL C02488 V=800.0 PL=0
MOVL C02489 V=800.0 PL=0
MOVL C02490 V=800.0 PL=0
MOVL C02491 V=800.0 PL=0
MOVL C02492 V=800.0 PL=0
MOVL C02493 V=800.0 PL=0
MOVL C02494 V=800.0 PL=0
MOVL C02495 V=800.0 PL=0
MOVL C02496 V=800.0 PL=0
MOVL C02497 V=800.0 PL=0
MOVL C02498 V=800.0 PL=0
MOVL C02499 V=800.0 PL=0
MOVL C02500 V=800.0 PL=0
MOVL C02501 V=800.0 PL=0
MOVL C02502 V=800.0 PL=0
MOVL C02503 V=800.0 PL=0
MOVL C02504 V=800.0 PL=0
MOVL C02505 V=800.0 PL=0
MOVL C02506 V=800.0 PL=0
MOVL C02507 V=800.0 PL=0
MOVL C02508 V=800.0 PL=0
MOVL C02509 V=800.0 PL=0
MOVL C02510 V=800.0 PL=0
MOVL C02511 V=800.0 PL=0
MOVL C02512 V=800.0 PL=0
MOVL C02513 V=800.0 PL=0
MOVL C02514 V=800.0 PL=0
MOVL C02515 V=800.0 PL=0
MOVL C02516 V=800.0 PL=0
MOVL C02517 V=800.0 PL=0
MOVL C02518 V=800.0 PL=0
MOVL C02519 V=800.0 PL=0
MOVL C02520 V=800.0 PL=0
MOVL C02521 V=800.0 PL=0
MOVL C02522 V=800.0 PL=0
MOVL C02523 V=800.0 PL=0
MOVL C02524 V=800.0 PL=0
MOVL C02525 V=800.0 PL=0
MOVL C02526 V=800.0 PL=0
MOVL C02527 V=800.0 PL=0
MOVL C02528 V=800.0 PL=0
MOVL C02529 V=800.0 PL=0
MOVL C02530 V=800.0 PL=0
MOVL C02531 V=800.0 PL=0
MOVL C02532 V=800.0 PL=0
MOVL C02533 V=800.0 PL=0
MOVL C02534 V=800.0 PL=0
MOVL C02535 V=800.0 PL=0
MOVL C02536 V=800.0 PL=0
MOVL C02537 V=800.0 PL=0
MOVL C02538 V=800.0 PL=0
MOVL C02539 V=800.0 PL=0
MOVL C02540 V=800.0 PL=0
MOVL C02541 V=800.0 PL=0
MOVL C02542 V=800.0 PL=0
MOVL C02543 V=800.0 PL=0
MOVL C02544 V=800.0 PL=0
MOVL C02545 V=800.0 PL=0
MOVL C02546 V=800.0 PL=0
MOVL C02547 V=800.0 PL=0
MOVL C02548 V=800.0 PL=0
MOVL C02549 V=800.0 PL=0
MOVL C02550 V=800.0 PL=0
MOVL C02551 V=800.0 PL=0
MOVL C02552 V=800.0 PL=0
MOVL C02553 V=800.0 PL=0
MOVL C02554 V=800.0 PL=0
MOVL C02555 V=800.0 PL=0
MOVL C02556 V=800.0 PL=0
MOVL C02557 V=800.0 PL=0
MOVL C02558 V=800.0 PL=0
MOVL C02559 V=800.0 PL=0
MOVL C02560 V=800.0 PL=0
MOVL C02561 V=800.0 PL=0
MOVL C02562 V=800.0 PL=0
MOVL C02563 V=800.0 PL=0
MOVL C02564 V=800.0 PL=0
MOVL C02565 V=800.0 PL=0
MOVL C02566 V=800.0 PL=0
MOVL C02567 V=800.0 PL=0
MOVL C02568 V=800.0 PL=0
MOVL C02569 V=800.0 PL=0
MOVL C02570 V=800.0 PL=0
MOVL C02571 V=800.0 PL=0
MOVL C02572 V=800.0 PL=0
MOVL C02573 V=800.0 PL=0
MOVL C02574 V=800.0 PL=0
MOVL C02575 V=800.0 PL=0
MOVL C02576 V=800.0 PL=0
MOVL C02577 V=800.0 PL=0
MOVL C02578 V=800.0 PL=0
MOVL C02579 V=800.0 PL=0
MOVL C02580 V=800.0 PL=0
MOVL C02581 V=800.0 PL=0
MOVL C02582 V=800.0 PL=0
MOVL C02583 V=800.0 PL=0
MOVL C02584 V=800.0 PL=0
MOVL C02585 V=800.0 PL=0
MOVL C02586 V=800.0 PL=0
MOVL C02587 V=800.0 PL=0
MOVL C02588 V=800.0 PL=0
MOVL C02589 V=800.0 PL=0
MOVL C02590 V=800.0 PL=0
MOVL C02591 V=800.0 PL=0
MOVL C02592 V=800.0 PL=0
MOVL C02593 V=800.0 PL=0
MOVL C02594 V=800.0 PL=0
MOVL C02595 V=800.0 PL=0
MOVL C02596 V=800.0 PL=0
MOVL C02597 V=800.0 PL=0
MOVL C02598 V=800.0 PL=0
MOVL C02599 V=800.0 PL=0
MOVL C02600 V=800.0 PL=0
MOVL C02601 V=800.0 PL=0
MOVL C02602 V=800.0 PL=0
MOVL C02603 V=800.0 PL=0
MOVL C02604 V=800.0 PL=0
MOVL C02605 V=800.0 PL=0
MOVL C02606 V=800.0 PL=0
MOVL C02607 V=800.0 PL=0
MOVL C02608 V=800.0 PL=0
MOVL C02609 V=800.0 PL=0
MOVL C02610 V=800.0 PL=0
MOVL C02611 V=800.0 PL=0
MOVL C02612 V=800.0 PL=0
MOVL C02613 V=800.0 PL=0
MOVL C02614 V=800.0 PL=0
MOVL C02615 V=800.0 PL=0
MOVL C02616 V=800.0 PL=0
MOVL C02617 V=800.0 PL=0
MOVL C02618 V=800.0 PL=0
MOVL C02619 V=800.0 PL=0
MOVL C02620 V=800.0 PL=0
MOVL C02621 V=800.0 PL=0
MOVL C02622 V=800.0 PL=0
MOVL C02623 V=800.0 PL=0
MOVL C02624 V=800.0 PL=0
MOVL C02625 V=800.0 PL=0
MOVL C02626 V=800.0 PL=0
MOVL C02627 V=800.0 PL=0
MOVL C02628 V=800.0 PL=0
MOVL C02629 V=800.0 PL=0
MOVL C02630 V=800.0 PL=0
MOVL C02631 V=800.0 PL=0
MOVL C02632 V=800.0 PL=0
MOVL C02633 V=800.0 PL=0
MOVL C02634 V=800.0 PL=0
MOVL C02635 V=800.0 PL=0
MOVL C02636 V=800.0 PL=0
MOVL C02637 V=800.0 PL=0
MOVL C02638 V=800.0 PL=0
MOVL C02639 V=800.0 PL=0
MOVL C02640 V=800.0 PL=0
MOVL C02641 V=800.0 PL=0
MOVL C02642 V=800.0 PL=0
MOVL C02643 V=800.0 PL=0
MOVL C02644 V=800.0 PL=0
MOVL C02645 V=800.0 PL=0
MOVL C02646 V=800.0 PL=0
MOVL C02647 V=800.0 PL=0
MOVL C02648 V=800.0 PL=0
MOVL C02649 V=800.0 PL=0
MOVL C02650 V=800.0 PL=0
MOVL C02651 V=800.0 PL=0
MOVL C02652 V=800.0 PL=0
MOVL C02653 V=800.0 PL=0
MOVL C02654 V=800.0 PL=0
MOVL C02655 V=800.0 PL=0
MOVL C02656 V=800.0 PL=0
MOVL C02657 V=800.0 PL=0
MOVL C02658 V=800.0 PL=0
MOVL C02659 V=800.0 PL=0
MOVL C02660 V=800.0 PL=0
MOVL C02661 V=800.0 PL=0
MOVL C02662 V=800.0 PL=0
MOVL C02663 V=800.0 PL=0
MOVL C02664 V=800.0 PL=0
MOVL C02665 V=800.0 PL=0
MOVL C02666 V=800.0 PL=0
MOVL C02667 V=800.0 PL=0
MOVL C02668 V=800.0 PL=0
MOVL C02669 V=800.0 PL=0
MOVL C02670 V=800.0 PL=0
MOVL C02671 V=800.0 PL=0
MOVL C02672 V=800.0 PL=0
MOVL C02673 V=800.0 PL=0
MOVL C02674 V=800.0 PL=0
MOVL C02675 V=800.0 PL=0
MOVL C02676 V=800.0 PL=0
MOVL C02677 V=800.0 PL=0
MOVL C02678 V=800.0 PL=0
MOVL C02679 V=800.0 PL=0
MOVL C02680 V=800.0 PL=0
MOVL C02681 V=800.0 PL=0
MOVL C02682 V=800.0 PL=0
MOVL C02683 V=800.0 PL=0
MOVL C02684 V=800.0 PL=0
MOVL C02685 V=800.0 PL=0
MOVL C02686 V=800.0 PL=0
MOVL C02687 V=800.0 PL=0
MOVL C02688 V=800.0 PL=0
MOVL C02689 V=800.0 PL=0
MOVL C02690 V=800.0 PL=0
MOVL C02691 V=800.0 PL=0
MOVL C02692 V=800.0 PL=0
MOVL C02693 V=800.0 PL=0
MOVL C02694 V=800.0 PL=0
MOVL C02695 V=800.0 PL=0
MOVL C02696 V=800.0 PL=0
MOVL C02697 V=800.0 PL=0
MOVL C02698 V=800.0 PL=0
MOVL C02699 V=800.0 PL=0
MOVL C02700 V=800.0 PL=0
MOVL C02701 V=800.0 PL=0
MOVL C02702 V=800.0 PL=0
